(* IEC 61131-3 sources: LASAL/Class/ST151Base, 1 file *)

(* ---- ST151Base.st ---- *)
#define DEVICE_ID_ST151                                                    1086

#define ST151_ADDR_PDO_WRITE                                            16#0000
#define ST151_ADDR_PDO_READ                                             16#0038
#define ST151_ADDR_SDO_1                                                16#0008
#define ST151_ADDR_SDO_2           (ST151_ADDR_SDO_1+sizeof(t_s_ConfigModule1))
#define ST151_ADDR_SDO_3                                (ST151_ADDR_PDO_READ+6)  //only read sdo!!!
#define ST151_ADDR_SDO_4           (ST151_ADDR_SDO_3+sizeof(t_s_ConfigModule3))
#define ST151_ADDR_SDO_5           (ST151_ADDR_SDO_4+sizeof(t_s_ConfigModule4))
#define ST151_ADDR_SDO_6           (ST151_ADDR_SDO_5+sizeof(t_s_ConfigModule5))

#define ST151_OSZI_ADDR_WRITE                                           16#0800
#define ST151_OSZI_ADDR_READ                                            16#0808
#define ST151_OSZI_ADDR_DATA                                            16#0820
#define ST151_OSZI_READPOINTER_OFFSET                                   16#0020
#define ST151_OSZI_ONE_PDOSIZE                                              126
#define ST151_OSZI_VALUES_DATA             (ST151_OSZI_ONE_PDOSIZE/sizeof(UINT))
#define ST151_OSZI_BUFFER_SIZE                                             1024
#define ST151_OSZI_MAX_SAMPLES             (ST151_OSZI_BUFFER_SIZE/sizeof(UINT))
#define ST151_OSZI_MAX_PDOREAD   ((ST151_OSZI_BUFFER_SIZE/ST151_OSZI_ONE_PDOSIZE)+1)

// in MHz
#define ST151_FREQUENCY_MHZ                             125
// in Hz
#define ST151_FREQUENCY_HZ   (ST151_FREQUENCY_MHZ * 1000000)

#define ST151_SDO_RESPONSE_TIMEOUT   (SDIAS_SDO_TIMEOUT * 2)
#define ST151_SDO_MAX_RETRYS                              3

#define ST151_MAXFREQUENCY_OUT                   2_000_000 // 2Mhz/64 max frequency of module output
#define ST151_MAXSTEPPING_MODES                          6
#define ST151_FREQLIMITS_TABLESIZE      (ST151_MAXSTEPPING_MODES*sizeof(UDINT)*2)

#define ST151_MAX_ALLOWED_PERCENT                      100 // maximum value for percent value
#define ST151_BLANKING_TIME                             10 // minimum on time of pwm (*20ns)

#define ST151_CYCLICREFRESHDATA_TIME                   200 // time to refresh asynchrone values
#define ST151_INVALID_VALUE                   16#8000_0010 // invalid value for server
#define ST151_AUTOSET_FREQUENCYLIMIT          16#0000_0000 // value for autoset limit
#define ST151_DEACTIVATE_FREQUENCYLIMIT       16#FFFF_FFFF // value for deactivate limit

#define ST151_MAX_ALLOWED_CURRENT                     5000 // max allowed current (5A) in mA, from h-bridge according to hw-documentation
#define ST151_MAX_ALLOWED_CHOPPEROFFTIME              2500 // max allowed chopper off time in 20ns steps
#define ST151_MIN_ALLOWED_CHOPPEROFFTIME              1500 // min allowed chopper off time in 20ns steps
#define ST151_STALL_CURRENT_LIMIT                     1000 // calculation for stall current in permille
#define ST151_CURRENTOFFSETADJUST_MAX                  250 // maximum current offset adjust in mA
#define ST151_CURRENTOFFSETADJUST_MIN                 -250 // minimum current offset adjust in mA

//pll settings
#define ST151_SYNC_OUT_ID                             16#03
#define ST151_PLL_OFFSET                             16#140
#define ST151_PLL_CONTROL               (ST151_PLL_OFFSET+8)

#define ST151_ERROR_BITMASK_STATE_WORD               0x013E
#define ST151_ERROR_BITMASK_EXTENDED_STATE_WORD      0xFF3E

(*!
<Class
	Name               = "ST151Base"
	Revision           = "1.2"
	RealtimeTask       = "false"
	CyclicTask         = "false"
	BackgroundTask     = "false"
	Sigmatek           = "true"
	OSInterface        = "false"
	HighPriority       = "false"
	Automatic          = "false"
	UpdateMode         = "Prescan"
	IconPath           = ".\Class\s-dias.ico"
	SharedCommandTable = "true"
	Objectsize         = "(910,120)"
	Comment            = "SDIAS Stepper Module (1x Motor Out max. 5A, 2x Digital In 24V, 2x STO Enable 24V, 1x Incremental Encoder Input, 1x Regen Resistor)">
	<Channels>
		<Server Name="ActPosition" Visualized="true" Initialize="false" WriteProtected="true" Retentive="false" Comment="Actual internal Step-Position as 64 micro step."/>
		<Server Name="ActRegenResistorLoad" Visualized="true" Initialize="false" WriteProtected="true" Retentive="false" Comment="Actual load of regen resistor in xxx [%].&#13;&#10;If the value is never refreshed it shows -2 147 483 632.&#13;&#10;- Value is read asynchronous"/>
		<Server Name="AxError" Visualized="true" Initialize="false" WriteProtected="true" Retentive="false" Comment="Shows a fault of power-stage.&#13;&#10;(eg. over temperature, over current, power not connected)"/>
		<Server Name="ChopperOffTime" Visualized="true" Initialize="true" DefValue="1562" WriteProtected="false" Retentive="false" Comment="Set fixed off-time of the PWM  [20ns steps].&#13;&#10;If the value is changed, it is transferred asynchronously to the module.&#13;&#10;Valid range is from 1500 up to 2500."/>
		<Server Name="ChopperOnTimeMin" Visualized="true" Initialize="true" DefValue="180" WriteProtected="false" Retentive="false" Comment="Set minimum on-time of the PWM  [20ns steps].&#13;&#10;If the value is changed, it is transferred asynchronously to the module.&#13;&#10;Valid range is from 0 up to 2500."/>
		<Server Name="ControlWord" Visualized="true" Initialize="false" WriteProtected="false" Retentive="false" Comment="SwitchOn + Enable: Enable Motor&#13;&#10;ResetFault: Quit Error&#13;&#10;Bit12 ManufactureSpec1: current increase allowed"/>
		<Server Name="CurrentIncrease" Visualized="true" Initialize="true" DefValue="1" WriteProtected="false" Retentive="false" Comment="allow sqrt(2) current increase in halfstep mode&#13;&#10;&#13;&#10;in microstep mode the increase is always active"/>
		<Server Name="CurrentOffsetAdjBridge1" Visualized="true" Initialize="true" DefValue="100" WriteProtected="false" Retentive="false" Comment="!This setting has no effect if the version of the module is &gt;= HW2.0X1.4!&#13;&#10;&#13;&#10;Set current offset adjustment for bridge in [mA].&#13;&#10;Valid range is from -250 to 250 and default value is 100."/>
		<Server Name="CurrentOffsetAdjBridge2" Visualized="true" Initialize="true" DefValue="100" WriteProtected="false" Retentive="false" Comment="!This setting has no effect if the version of the module is &gt;= HW2.0X1.4!&#13;&#10;&#13;&#10;Set current offset adjustment for bridge in [mA].&#13;&#10;Valid range is from -250 to 250 and default value is 100."/>
		<Server Name="Enable" Visualized="true" Initialize="false" WriteProtected="false" Retentive="false" Comment="Enable stepper output.&#13;&#10;0 .. disabled&#13;&#10;1 .. enabled"/>
		<Server Name="EnableSteps" Visualized="true" Initialize="true" DefValue="2#1000111" WriteProtected="false" Retentive="false" Comment="Enable or disable microstepping modes. The full step mode cannot be deactivated.&#13;&#10;Bit1 .. Fullstep mode&#13;&#10;Bit2 .. Halfstep mode&#13;&#10;Bit3 .. Microstepping mode 4&#13;&#10;Bit4 .. Microstepping mode 8&#13;&#10;Bit5 .. Microstepping mode 16&#13;&#10;Bit6 .. Microstepping mode 32&#13;&#10;Bit7 .. Microstepping mode 64"/>
		<Server Name="EncoderPosition" Visualized="true" Initialize="false" WriteProtected="true" Retentive="false" Comment="Actual position of encoder."/>
		<Server Name="ErrorInfo" Visualized="true" Initialize="false" WriteProtected="true" Retentive="false" Comment="Shows errors from hardware. Errors above Bit 16 are refreshed at cyclic task over &quot;RefreshValues&quot; server.&#13;&#10;Bit 1: reserved&#13;&#10;Bit 2: Fault (Bridge not ok)&#13;&#10;Bit 3: Temperature  not ok&#13;&#10;Bit 4: Over current&#13;&#10;Bit 5: STO switch off (en1/en2)&#13;&#10;Bit 6: STO test switch off (negative test during operation)&#13;&#10;Bit 7: reserved&#13;&#10;Bit 8: reserved&#13;&#10;Bit 9: Brake chopper over current (disable brake chopper) &#13;&#10;Bit 10: reserved&#13;&#10;Bit 11: reserved&#13;&#10;Bit 12: reserved&#13;&#10;Bit 13: reserved&#13;&#10;Bit 14: reserved&#13;&#10;Bit 15: reserved&#13;&#10;Bit 16: reserved&#13;&#10;&#13;&#10;refreshed asynchrone:&#13;&#10;Bit 17: Regen resistor load warning&#13;&#10;Bit 18: Over temperature warning&#13;&#10;Bit 19: Over temperature failure (disable drive)&#13;&#10;Bit 20: Over current failure GND (disable drive)&#13;&#10;Bit 21: Over current failure Bridge 1 (disable drive)&#13;&#10;Bit 22: Over current failure Bridge 2 (disable drive)&#13;&#10;Bit 23: Regen resistor load threshold bridge (disable bridge)&#13;&#10;Bit 24: Regen resistor load error threshold resistor (disable resistor)&#13;&#10;Bit 25: Bridge voltage too low&#13;&#10;Bit 26: Bridge voltage too high&#13;&#10;Bit 27: External Enable 1 (STO) not ok&#13;&#10;Bit 28: External Enable 2 (STO) not ok&#13;&#10;Bit 29: Safety start up status test not ok&#13;&#10;Bit 30: Motor enable error&#13;&#10;Bit 31: Three time sync in lost&#13;&#10;Bit 32: Safe Ramp down pending"/>
		<Server Name="ErrorQuit" Visualized="true" Initialize="false" WriteProtected="false" Retentive="false" Comment="quits error if server &quot;Error&quot; is set"/>
		<Server Name="ExtendedStateWord" Visualized="true" Initialize="false" WriteProtected="true" Retentive="false" Comment="Shows the extended motor state word.&#13;&#10;- Value is read asynchronous&#13;&#10;Bit 1 : Zero Position (Input)&#13;&#10;Bit 2 : Over temperature warning&#13;&#10;Bit 3 : Over temperature failure (disable drive)&#13;&#10;Bit 4 : Over current failure GND (disable drive)&#13;&#10;Bit 5 : Over current failure Bridge 1 (disable drive)&#13;&#10;Bit 6 : Over current failure Bridge 2 (disable drive)&#13;&#10;Bit 7 : 5V Incremental encoder ok&#13;&#10;Bit 8 : reserved&#13;&#10;Bit 9 : Bridge voltage too low&#13;&#10;Bit 10: Bridge voltage too high&#13;&#10;Bit 11: External Enable 1 (STO)&#13;&#10;Bit 12: External Enable 2 (STO)&#13;&#10;Bit 13: Safety start up status test ok&#13;&#10;Bit 14: Motor enable error&#13;&#10;Bit 15: Three time sync in lost&#13;&#10;Bit 16: Safe Ramp down pending"/>
		<Server Name="ExternalEnable1" Visualized="true" Initialize="false" WriteProtected="true" Retentive="false" Comment="State of External Enable  (STO).&#13;&#10;If the value is never refreshed it shows -2 147 483 632.&#13;&#10;- Value is read asynchronous&#13;&#10;0 .. off&#13;&#10;1 .. on&#13;&#10;"/>
		<Server Name="ExternalEnable2" Visualized="true" Initialize="false" WriteProtected="true" Retentive="false" Comment="State of External Enable  (STO).&#13;&#10;If the value is never refreshed it shows -2 147 483 632.&#13;&#10;- Value is read asynchronous&#13;&#10;0 .. off&#13;&#10;1 .. on&#13;&#10;"/>
		<Server Name="FastDecayTime" Visualized="true" Initialize="true" DefValue="200" WriteProtected="false" Retentive="false" Comment="Set Fast Decay time [20ns steps].&#13;&#10;If the value is changed, it is transferred asynchronously to the module.&#13;&#10;Must be smaller than chopper off time!"/>
		<Server Name="FastDecayTimeFallingStep" Visualized="true" Initialize="true" DefValue="600" WriteProtected="false" Retentive="false" Comment="Set Fast Decay time for falling step [20ns steps].&#13;&#10;If the value is changed, it is transferred asynchronously to the module.&#13;&#10;Must be smaller than chopper off time!"/>
		<Server Name="FrequLimitDecrease16to32" Visualized="true" Initialize="true" DefValue="0" WriteProtected="false" Retentive="false" Comment="Set Frequency stepping mode limit if frequence is decreased.&#13;&#10;If the value is changed, it is transferred asynchronously to the module.&#13;&#10;If value is set to 0 the limit is automatically set."/>
		<Server Name="FrequLimitDecrease1to2" Visualized="true" Initialize="true" DefValue="0" WriteProtected="false" Retentive="false" Comment="Set Frequency stepping mode limit if frequence is decreased.&#13;&#10;If the value is changed, it is transferred asynchronously to the module.&#13;&#10;If value is set to 0 the limit is automatically set."/>
		<Server Name="FrequLimitDecrease2to4" Visualized="true" Initialize="true" DefValue="0" WriteProtected="false" Retentive="false" Comment="Set Frequency stepping mode limit if frequence is decreased.&#13;&#10;If the value is changed, it is transferred asynchronously to the module.&#13;&#10;If value is set to 0 the limit is automatically set."/>
		<Server Name="FrequLimitDecrease32to64" Visualized="true" Initialize="true" DefValue="0" WriteProtected="false" Retentive="false" Comment="Set Frequency stepping mode limit if frequence is decreased.&#13;&#10;If the value is changed, it is transferred asynchronously to the module.&#13;&#10;If value is set to 0 the limit is automatically set."/>
		<Server Name="FrequLimitDecrease4to8" Visualized="true" Initialize="true" DefValue="0" WriteProtected="false" Retentive="false" Comment="Set Frequency stepping mode limit if frequence is decreased.&#13;&#10;If the value is changed, it is transferred asynchronously to the module.&#13;&#10;If value is set to 0 the limit is automatically set."/>
		<Server Name="FrequLimitDecrease8to16" Visualized="true" Initialize="true" DefValue="0" WriteProtected="false" Retentive="false" Comment="Set Frequency stepping mode limit if frequence is decreased.&#13;&#10;If the value is changed, it is transferred asynchronously to the module.&#13;&#10;If value is set to 0 the limit is automatically set."/>
		<Server Name="FrequLimitIncrease16to8" Visualized="true" Initialize="true" DefValue="20000" WriteProtected="false" Retentive="false" Comment="Set Frequency stepping mode limit if frequence is increased.&#13;&#10;If the value is changed, it is transferred asynchronously to the module.&#13;&#10;"/>
		<Server Name="FrequLimitIncrease2to1" Visualized="true" Initialize="true" DefValue="50000" WriteProtected="false" Retentive="false" Comment="Set Frequency stepping mode limit if frequence is increased.&#13;&#10;If the value is changed, it is transferred asynchronously to the module.&#13;&#10;"/>
		<Server Name="FrequLimitIncrease32to16" Visualized="true" Initialize="true" DefValue="10000" WriteProtected="false" Retentive="false" Comment="Set Frequency stepping mode limit if frequence is increased.&#13;&#10;If the value is changed, it is transferred asynchronously to the module.&#13;&#10;"/>
		<Server Name="FrequLimitIncrease4to2" Visualized="true" Initialize="true" DefValue="40000" WriteProtected="false" Retentive="false" Comment="Set Frequency stepping mode limit if frequence is increased.&#13;&#10;If the value is changed, it is transferred asynchronously to the module.&#13;&#10;"/>
		<Server Name="FrequLimitIncrease64to32" Visualized="true" Initialize="true" DefValue="5000" WriteProtected="false" Retentive="false" Comment="Set Frequency stepping mode limit if frequence is increased.&#13;&#10;If the value is changed, it is transferred asynchronously to the module.&#13;&#10;"/>
		<Server Name="FrequLimitIncrease8to4" Visualized="true" Initialize="true" DefValue="30000" WriteProtected="false" Retentive="false" Comment="Set Frequency stepping mode limit if frequence is increased.&#13;&#10;If the value is changed, it is transferred asynchronously to the module.&#13;&#10;"/>
		<Server Name="HBridgeTemperature" Visualized="true" Initialize="false" WriteProtected="true" Retentive="false" Comment="actual Temperature in xx.x [°C]&#13;&#10;If the value is never refreshed it shows -2 147 483 632.&#13;&#10;- Value is read asynchronous."/>
		<Server Name="HBridgeVoltage" Visualized="true" Initialize="false" WriteProtected="true" Retentive="false" Comment="Actual Voltage in xx.xx [V].&#13;&#10;If the value is never refreshed it shows -2 147 483 632.&#13;&#10;- Value is read asynchronous"/>
		<Server Name="HWEnableSoftwareRampdown" Visualized="true" Initialize="true" WriteProtected="false" Retentive="false" Comment=" 0 ... HardwareRampdown&#13;&#10; 1 ... SoftwareRampdown"/>
		<Server Name="HWRampdownDeltaFrequency" Visualized="true" Initialize="true" DefValue="40" WriteProtected="false" Retentive="false" Comment="If the enable-signal is lost the output frequency is decreased by HWRampdownDeltaFrequency every HWRampdownDeltaTime"/>
		<Server Name="HWRampdownDeltaTime" Visualized="true" Initialize="true" DefValue="1" WriteProtected="false" Retentive="false" Comment="[20ns steps]&#13;&#10;If the enable-signal is lost the output frequency is decreased by HWRampdownDeltaFrequency every HWRampdownDeltaTime"/>
		<Server Name="Input1" Visualized="true" Initialize="false" WriteProtected="true" Retentive="false" Comment="first digital input"/>
		<Server Name="Input1LatchedFalling" Visualized="true" Initialize="false" WriteProtected="true" Retentive="false" Comment="latched falling edge of first digital input&#13;&#10;signal will stay until read-method is called"/>
		<Server Name="Input1LatchedRising" Visualized="true" Initialize="false" WriteProtected="true" Retentive="false" Comment="latched rising edge of first digital input&#13;&#10;signal will stay until read-method is called"/>
		<Server Name="Input2" Visualized="true" Initialize="false" WriteProtected="true" Retentive="false" Comment="second digital input"/>
		<Server Name="Input2LatchedFalling" Visualized="true" Initialize="false" WriteProtected="true" Retentive="false" Comment="latched falling edge of second digital input&#13;&#10;signal will stay until read-method is called"/>
		<Server Name="Input2LatchedRising" Visualized="true" Initialize="false" WriteProtected="true" Retentive="false" Comment="latched rising edge of second digital input&#13;&#10;signal will stay until read-method is called"/>
		<Server Name="LatchPositionEncoderZeroPulse" Visualized="true" Initialize="false" WriteProtected="true" Retentive="false" Comment="Latched position of encoder zero pulse."/>
		<Server Name="LatchPositionInput1Falling" Visualized="true" Initialize="false" WriteProtected="true" Retentive="false" Comment="Latched position of falling edge of input 1."/>
		<Server Name="LatchPositionInput1Rising" Visualized="true" Initialize="false" WriteProtected="true" Retentive="false" Comment="Latched position of rising edge of input 1."/>
		<Server Name="LatchPositionInput2Falling" Visualized="true" Initialize="false" WriteProtected="true" Retentive="false" Comment="Latched position of falling edge of input 2."/>
		<Server Name="LatchPositionInput2Rising" Visualized="true" Initialize="false" WriteProtected="true" Retentive="false" Comment="Latched position of rising edge of input 2."/>
		<Server Name="MaxCurrent" Visualized="true" Initialize="true" WriteProtected="false" Retentive="false" Comment="Set maximum output current [mA] (effectiv value) as init value.&#13;&#10;If value is changed it is written asynchronosly.&#13;&#10;If the value is changed, it is transferred asynchronously to the module.&#13;&#10;Valid range is from 0 up to 5000."/>
		<Server Name="Online" Visualized="true" Initialize="false" WriteProtected="true" Retentive="false" Comment="Shows if hardware is ready.&#13;&#10;0 .. not ready&#13;&#10;1 .. ready"/>
		<Server Name="RefreshValues" Visualized="true" Initialize="true" WriteProtected="false" Retentive="false" Comment="Set refresh of asynchrone values&#13;&#10; 0 .. do not refresh values&#13;&#10; 1 .. do cyclic refresh of values (every 200ms)&#13;&#10; 2 .. refresh values once"/>
		<Server Name="SetFreqOut" Visualized="true" Initialize="false" WriteProtected="false" Retentive="false" Comment="Frequency in Hz of one Microstep [1/64 Hz]&#13;&#10;64 Microsteps = 1 Fullstep"/>
		<Server Name="StateWord" Visualized="true" Initialize="false" WriteProtected="true" Retentive="false" Comment="Statusword with DS402 Standard :&#13;&#10;Bit1  .. ReadyToSwitchOn&#13;&#10;Bit2  .. SwitchedOn&#13;&#10;Bit3  .. OperationEnabled&#13;&#10;Bit4  .. Fault&#13;&#10;Bit5  .. VoltageDisabled&#13;&#10;Bit6  .. QuickStop&#13;&#10;Bit7  .. SwitchOnDisabled&#13;&#10;Bit8  .. Warning&#13;&#10;Bit9  .. ManufactureSpecific1&#13;&#10;Bit10 .. Remote&#13;&#10;Bit11 .. TargetReached&#13;&#10;Bit12 .. InternalLimitActive&#13;&#10;Bit13 .. OperationModeSpecific1&#13;&#10;Bit14 .. OperationModeSpecific2&#13;&#10;Bit15 .. Manufacture Specific2&#13;&#10;Bit16 .. Manufacture Specific3"/>
		<Server Name="TargetFreqOut" Visualized="true" Initialize="false" WriteProtected="false" Retentive="false" Comment="Set desired motor frequency in [1/64 Hz].&#13;&#10;This value is needed for adaptive Microstepping calculation.&#13;&#10;64 Microsteps = 1 Fullstep&#13;&#10;-1 .. feature is deactivated."/>
		<Server Name="VoltageOKEncoder" Visualized="true" Initialize="false" WriteProtected="true" Retentive="false" Comment="Shows state of voltage supply of encoder.&#13;&#10;If the value is never refreshed it shows -2 147 483 632.&#13;&#10;- Value is read asynchronous&#13;&#10;0 .. Error at power supply.&#13;&#10;1 .. OK"/>
		<Server Name="ZPuls" Visualized="true" Initialize="false" WriteProtected="true" Retentive="false" Comment="It is 1 if incremental encoder zero position is passed."/>
		<Server Name="ZPulsLatched" Visualized="true" Initialize="false" WriteProtected="true" Retentive="false" Comment="It is 1 if incremental encoder zero position is passed, a read resets the server"/>
		<Client Name="ABCountMode" Required="true" Internal="false" DefValue="1" Comment="Set A/B count mode if &quot;1 edge&quot; sampling is activated, as init value.&#13;&#10;0 .. A pulses, B direction&#13;&#10;1 .. true A/B (default)"/>
		<Client Name="CompModeVST" Required="true" Internal="false" DefValue="0" Comment="Set Compatibility mode to VST01x as init value.&#13;&#10;0 .. Frequency as 64 microsteps - default&#13;&#10;1 .. Frequency as 32 microsteps&#13;&#10;This setting affects all &quot;FrequencyLimitsIncrease&quot;, &quot;FrequencyLimitsDecrease&quot;, &quot;SetFreqOut&quot;, &quot;ActPosition&quot;, &#13;&#10;&quot;TargetFreqOut&quot; server and the &quot;Latched Position&quot; server if LatchType is latch virtual counter."/>
		<Client Name="EnableRegenResistor" Required="true" Internal="false" DefValue="0" Comment="Enable external regen resistor.&#13;&#10;0 .. disabled&#13;&#10;1 .. enabled"/>
		<Client Name="EncMode" Required="true" Internal="false" DefValue="0" Comment="Mode of the Incremental Encoder as init value.&#13;&#10;0 .. TTL&#13;&#10;1 .. RS422&#13;&#10;"/>
		<Client Name="EncoderSampling" Required="true" Internal="false" DefValue="3" Comment="Sampling of the Incremental Encoder.&#13;&#10;0 .. Encoder off&#13;&#10;1 .. 1-edge&#13;&#10;2 .. 2-edge&#13;&#10;3 .. 4-edge&#13;&#10;"/>
		<Client Name="InvertEncoder" Required="true" Internal="false" DefValue="0" Comment="Counting direction of the encoder as initvalue.&#13;&#10;0 .. Phase B non-inverted&#13;&#10;1 .. Phase B inverted&#13;&#10;&#13;&#10;"/>
		<Client Name="InvertZeroPosition" Required="true" Internal="false" DefValue="0" Comment="Inverts server ZPulse as initvalue.&#13;&#10;0..normal &#13;&#10;1..inverted&#13;&#10;"/>
		<Client Name="LatchType" Required="true" Internal="false" DefValue="0" Comment="0 .. latch virtual counter&#13;&#10;1 .. latch incremental encoder&#13;&#10;as initvalue"/>
		<Client Name="LoadThresholdBridge" Required="true" Internal="false" DefValue="90" Comment="Set threshold value for regen resistor load [%] to switch off bridge, as init value.&#13;&#10;If this limit is reached, the bridge is switched off.&#13;&#10;Valid Range is 0 up to 100% and default value is 90%."/>
		<Client Name="LoadThresholdResistor" Required="true" Internal="false" DefValue="100" Comment="Set threshold value for regen resistor load [%] to switch external resistor off, as init value. &#13;&#10;If this limit is reached, the bridge and the regen resistor is switched off.&#13;&#10;Valid Range is 0 up to 100% and default value is 100%."/>
		<Client Name="LoadThresholdWarning" Required="true" Internal="false" DefValue="80" Comment="Set threshold value for regen resistor load [%] to set the warning bit, as init value.&#13;&#10;Valid Range is 0 up to 100% and default value is 80%."/>
		<Client Name="RatedMaxPower" Required="true" Internal="false" DefValue="1000" Comment="Set value for rated maximum Power of regen resistor in [1/10 W] as init value.&#13;&#10;Value is needed for capacity calculation of resistor.&#13;&#10;Valid range is from 1 up to 65535."/>
		<Client Name="RegenResistance" Required="true" Internal="false" DefValue="150" Comment="Set resistance of regen resistor in [1/10 Ohm] as init value.&#13;&#10;Value is needed for capacity calculation of resistor.&#13;&#10;Valid range is from 1 up to 65535."/>
		<Client Name="StallCurrentReduction" Required="true" Internal="false" DefValue="0" Comment="Value to reduce MaxCurrent for the Stop Position [0,1%] as init value. &#13;&#10;Defaultvalue: 0 (no reduction in the stop position)&#13;&#10;Range: 0 - 1000 (0-100%)&#13;&#10;Stop Position means, the value of the server SetFreqOut is lower than the StallCurrentWindow, &#13;&#10;which can be set with StallCurrentWindow and is 0 by default."/>
		<Client Name="StallCurrentWindow" Required="true" Internal="false" DefValue="0" Comment="Set a window in which the StallCurrentReduction setting is active as init value.&#13;&#10;Valid range is from 0 up to 65535."/>
		<Client Name="SteppingHysteresis" Required="true" Internal="false" DefValue="64" Comment="Set automatically stepping hysterese in [1/64 Hz] if the value for decrease limit is zero as init value.&#13;&#10;This value is substracted from the corresponding increase limit value and set for the decrease limit."/>
		<Client Name="toFreqLimitTable" Required="false" Internal="false"/>
		<Client Name="UseOszi" Required="true" Internal="false" DefValue="0" Comment="Activate oszi function of modul as init value.&#13;&#10;To use the Oszi function, the methods &quot;StartMeasure ()&quot; and &quot;GetMeasureState ()&quot; must be used.&#13;&#10;&#13;&#10;0 .. deactivated&#13;&#10;1 .. activated"/>
	</Channels>
	<Separators>
		<Servers>
			<SepChn Position="1"/>
			<SepChn Position="16"/>
			<SepChn Position="50"/>
		</Servers>
		<Clients>
			<SepChn Position="6"/>
		</Clients>
	</Separators>
	<RevDoku>
		<Owner Company="Sigmatek" Author="PieSte"/>
		<Dokumentation Revision="1.2" Date="31.07.2018" Author="RamAnd" Company="Sigmatek" Description="LASAL Hardware Description (.lhd) file has been updated.&#13;&#10;Removed initialize flag from server TargetFreqOut."/>
		<Dokumentation Revision="1.1" Date="01.02.2018" Author="ZoePat" Company="Sigmatek" Description="An error has been fixed if server settings were written in the init()."/>
		<Dokumentation Revision="1.0" Date="22.11.2017" Author="ZoePat" Company="Sigmatek" Description="first release version."/>
	</RevDoku>
	<Network Name="ST151Base">
		<!-- List of Components in this network -->
		<Components>
			<Object
				Name       = "_base"
				Class      = "SdiasBase"
				Position   = "(218,120)"
				Visualized = "true">
				<Channels>
					<Server Name="ClassState"/>
					<Server Name="DeviceID"/>
					<Server Name="FPGAVersion"/>
					<Server Name="HwVersion"/>
					<Server Name="LEDControl" Value="0"/>
					<Server Name="RetryCounter"/>
					<Server Name="SDOState"/>
					<Server Name="SerialNo"/>
					<Client Name="Place" Value="0"/>
					<Client Name="Required" Value="1"/>
					<Client Name="SdiasIn"/>
					<Client Name="ToStdLib"/>
				</Channels>
			</Object>
		</Components>
		<Comments>
		</Comments>
		<!-- List of Connections in this network -->
		<Connections>
			<Connection Source="this.ClassState" Destination="_base.ClassState" Vertices="(804,210),(632,210),"/>
			<Connection Source="this.DeviceID" Destination="_base.DeviceID" Vertices="(804,270),(632,270),"/>
			<Connection Source="this.FPGAVersion" Destination="_base.FPGAVersion" Vertices="(804,330),(632,330),"/>
			<Connection Source="this.SerialNo" Destination="_base.SerialNo" Vertices="(804,450),(632,450),"/>
			<Connection Source="this.RetryCounter" Destination="_base.RetryCounter" Vertices="(804,510),(632,510),"/>
			<Connection Source="this.LEDControl" Destination="_base.LEDControl" Vertices="(804,570),(632,570),"/>
			<Connection Source="_base.SdiasIn" Destination="this.SdiasIn" Vertices="(218,210),(38,210),"/>
			<Connection Source="_base.Place" Destination="this.Place" Vertices="(218,270),(38,270),"/>
			<Connection Source="_base.Required" Destination="this.Required" Vertices="(218,330),(38,330),"/>
			<Connection Source="this.HwVersion" Destination="_base.HwVersion" Vertices="(804,390),(632,390),"/>
			<Connection Source="this.SDOState" Destination="_base.SDOState" Vertices="(804,630),(632,630),"/>
		</Connections>
		<!-- Headerfiles -->
		<Options>
		</Options>
	</Network>
</Class>
*)
#pragma using SdiasBase

ST151Base : CLASS
: SdiasBase
	TYPE
	  a_uiOsziValues : ARRAY [0..ST151_OSZI_VALUES_DATA-1] OF UINT;
	  bd_EnabledFreqLimit : BDINT  //! <Type Public="true" Name="bd_EnabledFreqLimit"/>
	  [
	    1 FullStep,
	    2 HalfStep,
	    3 MicroStepping4,
	    4 MicroStepping8,
	    5 MicroStepping16,
	    6 MicroStepping32,
	    7 MicroStepping64,
	    8 Bit8,
	    9 Bit9,
	    10 Bit10,
	    11 Bit11,
	    12 Bit12,
	    13 Bit13,
	    14 Bit14,
	    15 Bit15,
	    16 Bit16,
	    17 Bit17,
	    18 Bit18,
	    19 Bit19,
	    20 Bit20,
	    21 Bit21,
	    22 Bit22,
	    23 Bit23,
	    24 Bit24,
	    25 Bit25,
	    26 Bit26,
	    27 Bit27,
	    28 Bit28,
	    29 Bit29,
	    30 Bit30,
	    31 Bit31,
	    32 Bit32,
	  ];
	  bd_ExtendedStateWord : BDINT  //! <Type Public="true" Name="bd_ExtendedStateWord"/>
	  [
	    1 ZeroPosition,
	    2 OverTempWarning,
	    3 OverTempFailure,
	    4 OverCurrentFailureGND,
	    5 OverCurrentFailureBridge1,
	    6 OverCurrentFailureBridge2,
	    7 Encoder5VOk,
	    8 Bit8,
	    9 BridgeVoltageTooLow,
	    10 BridgeVoltageTooHigh,
	    11 ExternEnableSTO1,
	    12 ExternEnableSTO2,
	    13 SafetyStartUpOK,
	    14 MotorEnableError,
	    15 ThreeTimeSyncInLost,
	    16 SafeRampDownPending,
	    17 LoadWarning,
	    18 LoadDisableBridge,
	    19 LoadDisableResistor,
	    20 Bit20,
	    21 Bit21,
	    22 Bit22,
	    23 Bit23,
	    24 Bit24,
	    25 Bit25,
	    26 Bit26,
	    27 Bit27,
	    28 Bit28,
	    29 Bit29,
	    30 Bit30,
	    31 Bit31,
	    32 Bit32,
	  ];
	  e_ActStepMode :
	  (
	    Microstepping_1,
	    Microstepping_2,
	    Microstepping_4,
	    Microstepping_8,
	    Microstepping_16,
	    Microstepping_32,
	    Microstepping_64
	  )$UDINT;
	  t_StatusWord : BINT
	  [
	    1 MotorEnabled,
	    2 Fault,
	    3 TemperatureOk,
	    4 OverCurrent,
	    5 STOSwitchOff,
	    6 STOTestSwitchOff,
	    7 STOReadyRestart,
	    8 ReadyToSwitchOn,
	    9 BrakeChopperOverCurrentLatch,
	    10 LatchIncZero,
	    11 LatchDigIn1Rise,
	    12 LatchDigIn1Fall,
	    13 LatchDigIn2Rise,  //! <Type Comment="Low bit of failure state depending on InternalLimitActive bit&#13;&#10;&#13;&#10;Meaning:&#13;&#10;2#00...No failure&#13;&#10;2#01...Overtemperature failure&#13;&#10;2#10...Overcurrent failure" Name="t_StatusWord.LatchDigIn2Rise"/>
	    14 LatchDigIn2Fall,  //! <Type Comment="High bit of failure state depending on InternalLimitActive bit&#13;&#10;&#13;&#10;Meaning:&#13;&#10;2#00...No failure&#13;&#10;2#01...Overtemperature failure&#13;&#10;2#10...Overcurrent failure" Name="t_StatusWord.LatchDigIn2Fall"/>
	    15 DigIn1,  //! <Type Comment="Low bit of failure state depending on InternalLimitActive bit&#13;&#10;&#13;&#10;Meaning:&#13;&#10;2#00...No failure&#13;&#10;2#01...Overtemperature failure&#13;&#10;2#10...Overcurrent failure" Name="t_StatusWord.DigIn1"/>
	    16 DigIn2,  //! <Type Comment="High bit of failure state depending on InternalLimitActive bit&#13;&#10;&#13;&#10;Meaning:&#13;&#10;2#00...No failure&#13;&#10;2#01...Overtemperature failure&#13;&#10;2#10...Overcurrent failure" Name="t_StatusWord.DigIn2"/>
	  ];
#pragma pack(push, 1)
	  t_s_ReadData : STRUCT
	    StateWord : t_StatusWord;
	    ActPos : UINT;
	    IncrementalEncoderValue : UINT;
	  END_STRUCT;
#pragma pack(pop)
	  t_ControlWord : BINT
	  [
	    1 SwitchOn,
	    2 FaultReset,
	    3 CurrentDropEnable,
	    4 CurrentIncrease,
	    5 HWEnableSofwareRampdownToggleBit,
	    6 QuitSTOOff,
	    7 RegenResistorEnable,
	    8 RegenResistorFaultReset,
	    9 SwitchMaxCurrent,  //! <Type Comment="0 .. internal counter&#13;&#10;1 .. incremental encoder" Name="t_ControlWord.SwitchMaxCurrent"/>
	    10 EnableStep64,
	    11 EnableStep32,
	    12 EnableStep16,
	    13 EnableStep8,
	    14 EnableStep4,
	    15 EnableHalfStep,
	    16 EnableFullStep,
	  ];
#pragma pack(push, 1)
	  t_s_WriteData : STRUCT
	    StepFrequencyReg : DINT;
	    ControlWord : t_ControlWord;
	  END_STRUCT;
#pragma pack(pop)
#pragma pack(push, 1)
	  t_Accesses : STRUCT
	    pReadData : ^t_s_ReadData;
	    pWriteData : ^t_s_WriteData;
	    sWriteData : t_s_WriteData;
	  END_STRUCT;
#pragma pack(pop)
#pragma pack(push, 1)
	  t_s_ControlAccess : STRUCT
	    AccessHandle : UDINT;
	    pControlByte : t_SDIAS_pControlByte;
	    pStateByte : t_SDIAS_pStateByte;
	  END_STRUCT;
#pragma pack(pop)
#pragma pack(push, 1)
	  t_s_OsziWrite : STRUCT
	    SamplesAfterTrigger : UINT;
	    TriggerLevel : UINT;
	    SampleTimePrescaler : UINT;
	    TriggerChannelSelect : USINT;
	    ControlOszi : BSINT
	    [
	      1 StartTriggering,
	      2 CancelTrigger,
	      3 RisingEdge,
	      4 FallingEdge,
	      5 Force,
	      6 Bit6,
	      7 Bit7,
	      8 Bit8,
	    ];
	  END_STRUCT;
#pragma pack(pop)
#pragma pack(push, 1)
	  t_s_OsziRead : STRUCT
	    SizeOfRam : UDINT;
	    PointerOnLastSampleData : HDINT;
	    StateOszi : BSINT
	    [
	      1 Ready,
	      2 Triggered,
	      3 BufferOverflow,
	      4 Bit4,
	      5 Bit5,
	      6 Bit6,
	      7 Bit7,
	      8 Bit8,
	    ];
	    NbrOfChAvailable : USINT;
	  END_STRUCT;
#pragma pack(pop)
#pragma pack(push, 1)
	  t_AccessesOszi : STRUCT
	    WriteHeaderControl : t_s_ControlAccess;
	    pWriteHeader : ^t_s_OsziWrite;
	    sWriteOszi : t_s_OsziWrite;
	    ReadHeaderControl : t_s_ControlAccess;
	    pReadHeader : ^t_s_OsziRead;
	    aReadDataControl : ARRAY [0..ST151_OSZI_MAX_PDOREAD-1] OF t_s_ControlAccess;
	    apOsziData : ARRAY [0..ST151_OSZI_MAX_PDOREAD-1] OF ^a_uiOsziValues;
	    uiSamplesAfterTrigger : UINT;
	    uiSamplesBeforeTrigger : UINT;
	    bDataReady : DINT;
	    bSplitBuffer : BOOL;
	    uiDatalength1 : UINT;
	    uiDatalength2 : UINT;
	    eOsziData :
	    (
	      _OsziDataIdle,
	      _OsziTriggerStart,
	      _OsziResetTrigger,
	      _OsziWait4Reset,
	      _OsziWait4Trigger,
	      _OsziDisableRead,
	      _OsziGetData,
	      _OsziWait4Data,
	      _OsziFinished
	    )$UDINT;
	    sLastOsziState : t_s_OsziRead;
	    aLastOsziData : ARRAY [0..ST151_OSZI_MAX_SAMPLES-1] OF UINT;
	    pLastEntryOsziData : ^UINT;
	    pFirstEntryOsziData : ^UINT;
	    pToExternData : ^void;
	    usOsziTriggerOffset : USINT;
	    bMeasureStarted : BOOL;
	  END_STRUCT;
#pragma pack(pop)
	  t_bi_ReqSDOConfig : BINT
	  [
	    1 WriteConfigSDO1,
	    2 WriteConfigSDO2,
	    3 WriteConfigSDO3,
	    4 WriteConfigSDO4,
	    5 WriteConfigSDO5,
	    6 WriteConfigSDO6,
	    7 Bit7,
	    8 ReadConfigSDO1,
	    9 ReadConfigSDO2,
	    10 ReadConfigSDO3,
	    11 ReadConfigSDO4,
	    12 ReadConfigSDO5,
	    13 ReadConfigSDO6,
	    14 Bit14,
	    15 Bit15,
	    16 Bit16,
	  ];
	  t_bs_IsyncValue : BSINT
	  [
	    1 IncZero,
	    2 DigIn1Rise,
	    3 DigIn1Fall,
	    4 DigIn2Rise,
	    5 DigIn2Fall,
	  ];
	  t_e_InitSSW :
	  (
	    _ReadInitValuesFromModule,
	    _InitVariables,
	    _WriteConfigSDO,
	    _ReadConfigSDO,
	    _DisablePll,
	    _ReadPll,
	    _SetPll,
	    _Wait4FPGAReset,
	    _ActivateFPGA,
	    _Finish,
	    _InitError
	  )$UDINT;
	  t_e_SDOConfig :
	  (
	    _SDOConfig_Idle,
	    _SDOConfig_Write1,
	    _SDOConfig_Write2,
	    _SDOConfig_Write3,
	    _SDOConfig_Write4,
	    _SDOConfig_Write5,
	    _SDOConfig_Write6,
	    _SDOConfig_Read1,
	    _SDOConfig_Read2,
	    _SDOConfig_Read3,
	    _SDOConfig_Read4,
	    _SDOConfig_Read5,
	    _SDOConfig_Read6,
	    _SDOConfig_Finished,
	    _SDOConfig_Error
	  )$UDINT;
#pragma pack(push, 1)
	  t_EnabledFreqLimit : STRUCT
	    DecreaseFreq : bd_EnabledFreqLimit;
	    IncreaseFreq : bd_EnabledFreqLimit;
	  END_STRUCT;
#pragma pack(pop)
#pragma pack(push, 1)
	  t_FrequencyLimits : STRUCT
	    LimitDecrease : UDINT;  //! <Type Comment="save the higher limit" Name="t_FrequencyLimits.LimitDecrease"/>
	    LimitIncrease : UDINT;  //! <Type Comment="save the lower limit" Name="t_FrequencyLimits.LimitIncrease"/>
	  END_STRUCT;
#pragma pack(pop)
#pragma pack(push, 1)
	  t_LatchValues : STRUCT
	    uiISyncIncZeroOldCounter : UINT;
	    uiISyncDigIn1RiseOldCounter : UINT;
	    uiISyncDigIn1FallOldCounter : UINT;
	    uiISyncDigIn2RiseOldCounter : UINT;
	    uiISyncDigIn2FallOldCounter : UINT;
	    sdISyncIncZeroOldPosition : DINT;
	    sdISyncDigIn1RiseOldPosition : DINT;
	    sdISyncDigIn1FallOldPosition : DINT;
	    sdISyncDigIn2RiseOldPosition : DINT;
	    sdISyncDigIn2FallOldPosition : DINT;
	    uiLatchInputZero : DINT;
	    uiLatchInputDigIn1Rising : UINT;
	    uiLatchInputDigIn1Falling : UINT;
	    uiLatchInputDigIn2Rising : UINT;
	    uiLatchInputDigIn2Falling : UINT;
	    bsValidISyncValue : t_bs_IsyncValue;
	    bsActiveISyncValue : t_bs_IsyncValue;
	    bsLatchReaded : t_bs_IsyncValue;
	    bResetActiveSyncValue : BOOL;
	  END_STRUCT;
#pragma pack(pop)
#pragma pack(push, 1)
	  t_SyncOut : STRUCT
	    uiOffset : UINT;
	    usPeriodMulti : USINT;
	    bsSyncStartDelay : BSINT
	    [
	      1 SyncStartDelay1,
	      2 SyncStartDelay2,
	      3 SyncStartDelay3,
	      4 SyncStartDelay4,
	    ];
	    hsSyncOutID : HSINT;
	    bsControlState : BSINT
	    [
	      1 SyncEnable,
	      2 StartDelayEnable,
	      3 SyncSelector,
	    ];
	    uiReserved : UINT;
	  END_STRUCT;
#pragma pack(pop)
#pragma pack(push, 1)
	  t_PllRegister : STRUCT
	    udSystemPerTime : UDINT;
	    udSystemPerTimeMeasure : UDINT;
	    bsStateControlReg : BSINT
	    [
	      1 locked_res1,
	      2 unlocked_res2,
	      3 Soft_enable,
	      4 res3,
	      5 res4,
	      6 res5,
	      7 res6,
	      8 res7,
	    ];
	    usSystemPeriodeDividier : USINT;
	    bsCompDelay : BSINT
	    [
	    ];
	    usReserved : USINT;
	    SyncOut0 : t_SyncOut;
	  END_STRUCT;
#pragma pack(pop)
	  t_ResponseState :
	  (
	    _idle,
	    _wait,
	    _valid
	  )$UDINT;
#pragma pack(push, 1)
	  t_s_AdaptiveSteppingCalc : STRUCT
	    usIncreaseActStepsActivated : USINT;
	    aIncreaseLimitsArrayEntry : ARRAY [0..ST151_MAXSTEPPING_MODES] OF USINT;
	    usDecreaseActStepsActivated : USINT;
	    aDecreaseLimitsArrayEntry : ARRAY [0..ST151_MAXSTEPPING_MODES] OF USINT;
	  END_STRUCT;
#pragma pack(pop)
#pragma pack(push, 1)
	  t_s_ConfigModule1 : STRUCT
	    ChopperOffTime : UINT;
	    FastDecayTime : UINT;
	    FrequLimitRising64 : UDINT;
	    FrequLimitRising32 : UDINT;
	    FrequLimitRising16 : UDINT;
	    FrequLimitRising8 : UDINT;
	    FrequLimitRising4 : UDINT;
	    FrequLimitRising2 : UDINT;
	  END_STRUCT;
#pragma pack(pop)
#pragma pack(push, 1)
	  t_s_ConfigModule2 : STRUCT
	    HWRampdownDeltaFrequency : UINT;
	    HWRampdownDeltaTime : UINT;
	    IncrementalEncoderSettings : BSINT
	    [
	      1 ZeroPosInversion,
	      2 PhaseBInversion,
	      3 EdgeSampling1,
	      4 EdgeSampling2,
	      5 TTL_RS422Mode,
	      6 ABCountMode,
	      7 LatchType,
	      8 Bit8,
	    ];
	    BlankingTimeRegister : USINT;
	    reserved1 : USINT;
	    reserved2 : USINT;
	    RatedMaximumPowerWatt : UINT;
	    RegenResistance : UINT;
	    LoadThresholdWarning : USINT;
	    LoadThresholdDisableResistor : USINT;
	    MaximumCurrentReg : UINT;
	    ReducedCurrentReg : UINT;
	    LoadThresholdDisableBridge : USINT;
	  END_STRUCT;
#pragma pack(pop)
#pragma pack(push, 1)
	  t_s_ConfigModule3 : STRUCT
	    LatchCntZPuls : UINT;
	    LatchCntInput1Rising : UINT;
	    LatchCntInput1Falling : UINT;
	    LatchCntInput2Rising : UINT;
	    LatchCntInput2Falling : UINT;
	  END_STRUCT;
#pragma pack(pop)
#pragma pack(push, 1)
	  t_s_ConfigModule4 : STRUCT
	    ExtendedMotorStateReg1 : BINT
	    [
	      1 ZeroPosition,
	      2 OverTempWarning,
	      3 OverTempFailure,
	      4 OverCurrentFailureGND,
	      5 OverCurrentFailureBridge1,
	      6 OverCurrentFailureBridge2,
	      7 Encoder5VOk,
	      8 Bit8,
	      9 BridgeVoltageTooLow,
	      10 BridgeVoltageTooHigh,
	      11 ExternEnableSTO1,
	      12 ExternEnableSTO2,
	      13 SafetyStartUpOK,
	      14 MotorEnableError,
	      15 ThreeTimeSyncInLost,
	      16 SafeRampDownPending,
	    ];
	    ExtendedMotorStateReg2 : BSINT
	    [
	      1 LoadWarning,
	      2 LoadDisableBridge,
	      3 LoadDisableResistor,
	    ];
	    ActRegenResistorLoad : USINT;
	    u2tValue : UDINT;
	    HBridgeVoltage : INT;
	    HBridgeTemperature : INT;
	    CommutationCntHBridge1 : UINT;
	    CommutationCntHBridge2 : UINT;
	    OntimeCntHBridge1 : UINT;
	    OntimeCntHBridge2 : UINT;
	    bsControllerStateReg : BSINT
	    [
	      1 NoCalibData,
	      2 InvalidCalibData,
	      3 Bit3,
	      4 ControllerOP,
	      5 Bit5,
	      6 Bit6,
	      7 Bit7,
	      8 Bit8,
	    ];
	  END_STRUCT;
#pragma pack(pop)
#pragma pack(push, 1)
	  t_s_ConfigModule5 : STRUCT
	    bsControllerControlReg : BSINT
	    [
	      1 Bit1,
	      2 Bit2,
	      3 Bit3,
	      4 Bit4,
	      5 Bit5,
	      6 Bit6,
	      7 LoadConfigNew,
	      8 ControllerReset,
	    ];
	    reserved1 : UINT;
	    FrequLimitFalling32to64 : UDINT;
	    FrequLimitFalling16to32 : UDINT;
	    FrequLimitFalling8to16 : UDINT;
	    FrequLimitFalling4to8 : UDINT;
	    FrequLimitFalling2to4 : UDINT;
	    FrequLimitFalling1to2 : UDINT;
	    FastDecayTimeFallingStep : UINT;
	    ChopperOnTimeMin : UINT;
	  END_STRUCT;
#pragma pack(pop)
#pragma pack(push, 1)
	  t_s_ConfigModule6 : STRUCT
	    CurrentOffsetAdjBridge1 : INT;
	    CurrentOffsetAdjBridge2 : INT;
	  END_STRUCT;
#pragma pack(pop)
#pragma pack(push, 1)
	  t_s_ConfigModul : STRUCT
	    SDOData1 : t_s_ConfigModule1;
	    SDOData2 : t_s_ConfigModule2;
	    SDOData3 : t_s_ConfigModule3;
	    SDOData4 : t_s_ConfigModule4;
	    SDOData5 : t_s_ConfigModule5;
	    SDOData6 : t_s_ConfigModule6;
	  END_STRUCT;
#pragma pack(pop)
#pragma pack(push, 1)
	  t_SPI_CalibHeader : STRUCT
	    ud_Checksum : UDINT;
	    ud_ListVersion : UDINT;
	    ud_ListLength : UDINT;
	  END_STRUCT;
#pragma pack(pop)
#pragma pack(push, 1)
	  t_SPI_CalibData : STRUCT
	    SPI_Header : t_SPI_CalibHeader;
	    Offset0 : INT;
	    Multiplier0 : INT;
	    Divisor0 : UINT;
	    Offset1 : INT;
	    Multiplier1 : INT;
	    Divisor1 : UINT;
	    AI1Offset : INT;
	    AI1Multiplikator : INT;
	    AI1Divisor : INT;
	    AI2Offset : INT;
	    AI2Multiplikator : INT;
	    AI2Divisor : INT;
	    BridgeMaximumCurrent : UINT;
	    BridgeSupplyVoltageLowerThreshold : UINT;
	    BridgeSupplyVoltageUpperThreshold : UINT;
	    BridgeTemperatureWarningThreshold : UINT;
	    BridgeTemperatureErrorThreshold : UINT;
	  END_STRUCT;
#pragma pack(pop)
#pragma pack(push, 1)
	  t_SPIReadData : STRUCT
	    IDHeader : t_SPI_ListHeader;
	    udMaxDataLength : UDINT;
	    udActReadLength : UDINT;
	    udReadLength : UDINT;
	    udReadOffset : UDINT;
	  END_STRUCT;
#pragma pack(pop)
#pragma pack(push, 1)
	  t_SPIWriteData : STRUCT
	    usBytesToWrite : USINT;
	    usBytesActWrite : USINT;
	    usWriteOffset : USINT;
	  END_STRUCT;
#pragma pack(pop)
	END_TYPE
  //Servers:
	Online 	: SvrCh_DINT;
	EncoderPosition 	: SvrCh_DINT;
	ZPuls 	: SvrCh_DINT;
	ZPulsLatched 	: SvrCh_DINT;
	LatchPositionEncoderZeroPulse 	: SvrCh_DINT;
	LatchPositionInput1Rising 	: SvrCh_DINT;
	LatchPositionInput1Falling 	: SvrCh_DINT;
	LatchPositionInput2Rising 	: SvrCh_DINT;
	LatchPositionInput2Falling 	: SvrCh_DINT;
	Input1 	: SvrCh_DINT;
	Input1LatchedRising 	: SvrCh_DINT;
	Input1LatchedFalling 	: SvrCh_DINT;
	Input2 	: SvrCh_DINT;
	Input2LatchedRising 	: SvrCh_DINT;
	Input2LatchedFalling 	: SvrCh_DINT;
	Enable 	: SvrCh_DINT;
	ActPosition 	: SvrCh_DINT;
	SetFreqOut 	: SvrCh_DINT;
	TargetFreqOut 	: SvrCh_DINT;
	CurrentIncrease 	: SvrCh_DINT;
	ControlWord 	: SvrCh_DS402_Control;
	StateWord 	: SvrCh_DS402_State;
	ErrorInfo 	: SvrCh_BDINT;
	AxError 	: SvrCh_DINT;
	ErrorQuit 	: SvrCh_DINT;
	HWEnableSoftwareRampdown 	: SvrCh_DINT;
	HWRampdownDeltaFrequency 	: SvrCh_DINT;
	HWRampdownDeltaTime 	: SvrCh_DINT;
	MaxCurrent 	: SvrCh_DINT;
	CurrentOffsetAdjBridge1 	: SvrCh_DINT;
	CurrentOffsetAdjBridge2 	: SvrCh_DINT;
	ChopperOffTime 	: SvrCh_DINT;
	ChopperOnTimeMin 	: SvrCh_DINT;
	FastDecayTime 	: SvrCh_DINT;
	FastDecayTimeFallingStep 	: SvrCh_DINT;
	EnableSteps 	: SvrCh_bd_EnabledFreqLimit_PTofCls_ST151Base;
	FrequLimitIncrease2to1 	: SvrCh_UDINT;
	FrequLimitIncrease4to2 	: SvrCh_UDINT;
	FrequLimitIncrease8to4 	: SvrCh_UDINT;
	FrequLimitIncrease16to8 	: SvrCh_UDINT;
	FrequLimitIncrease32to16 	: SvrCh_UDINT;
	FrequLimitIncrease64to32 	: SvrCh_UDINT;
	FrequLimitDecrease1to2 	: SvrCh_UDINT;
	FrequLimitDecrease2to4 	: SvrCh_UDINT;
	FrequLimitDecrease4to8 	: SvrCh_UDINT;
	FrequLimitDecrease8to16 	: SvrCh_UDINT;
	FrequLimitDecrease16to32 	: SvrCh_UDINT;
	FrequLimitDecrease32to64 	: SvrCh_UDINT;
	RefreshValues 	: SvrCh_DINT;
	ExtendedStateWord 	: SvrCh_bd_ExtendedStateWord_PTofCls_ST151Base;
	HBridgeVoltage 	: SvrChCmd_DINT;
	HBridgeTemperature 	: SvrCh_DINT;
	ExternalEnable1 	: SvrCh_DINT;
	ExternalEnable2 	: SvrCh_DINT;
	ActRegenResistorLoad 	: SvrCh_DINT;
	VoltageOKEncoder 	: SvrCh_DINT;
  //Clients:
	InvertEncoder 	: CltCh_DINT;
	InvertZeroPosition 	: CltCh_DINT;
	EncoderSampling 	: CltCh_DINT;
	EncMode 	: CltCh_DINT;
	LatchType 	: CltCh_DINT;
	ABCountMode 	: CltCh_DINT;
	StallCurrentReduction 	: CltCh_DINT;
	StallCurrentWindow 	: CltCh_DINT;
	EnableRegenResistor 	: CltCh_DINT;
	RegenResistance 	: CltCh_DINT;
	RatedMaxPower 	: CltCh_DINT;
	LoadThresholdWarning 	: CltCh_DINT;
	LoadThresholdBridge 	: CltCh_DINT;
	LoadThresholdResistor 	: CltCh_DINT;
	SteppingHysteresis 	: CltCh_DINT;
	CompModeVST 	: CltCh_DINT;
	UseOszi 	: CltCh_DINT;
	toFreqLimitTable 	: CltCh_DINT;
  //Variables:
		sAccesses 	: t_Accesses;
		sAccessesOszi 	: t_AccessesOszi;
		eActStepping 	: e_ActStepMode;
		sWriteSDO 	: t_s_ConfigModul;
		sReadSDO 	: t_s_ConfigModul;
		udStallCurrentWindow 	: UDINT;
		uiPositionOld 	: UINT;
		eInitSSW 	: t_e_InitSSW;
		eInitSSWErrorStep 	: t_e_InitSSW;
		eResponseState 	: t_ResponseState;
		udSDOTimeOut 	: UDINT;
		aFrequencyLimit : ARRAY [0..ST151_MAXSTEPPING_MODES] OF t_FrequencyLimits;

		eActSDOConfigRdWr 	: t_e_SDOConfig;
		biReqSDOConfigRdWr 	: t_bi_ReqSDOConfig;
		bsRespSDOConfigRdWr 	: t_bi_ReqSDOConfig;
		usSDORetrys 	: USINT;
		uiOldCntVirtual 	: UINT;
		uiOldCntEncoder 	: UINT;
		sPLLRegister 	: t_PllRegister;
		sSPIReadData 	: t_SPIReadData;
		sSPIWriteData 	: t_SPIWriteData;
		sStepsNeeded 	: t_EnabledFreqLimit;
		dActDirection 	: DINT;
		dOldSetFrequ 	: DINT;
		udCyclicRefresh 	: UDINT;
		dFrequBandwith 	: DINT;
		dHighFrequencyLimit 	: DINT;
		sAdaptiveStepping 	: t_s_AdaptiveSteppingCalc;
		sLatchValues 	: t_LatchValues;
		udStartWaitTime 	: UDINT;
		udLimitsHysteresis 	: UDINT;
		usCompModeVST 	: USINT;
  //Functions:
				//! <Function Comment="Init-Methode of Class.&#13;&#10;&#13;&#10;This Methode needs to get called. In case the Methode gets overwritten, a call needs to bet installed." Name="Init"/>
	FUNCTION VIRTUAL GLOBAL Init;

	FUNCTION ST151Base
		VAR_OUTPUT
			ret_code 	: ConfStates;
		END_VAR;
				//! <Function Comment="Realtime Update Methode which runs in PreScan." Name="UpdateRt"/>
	FUNCTION VIRTUAL GLOBAL UpdateRt;
				//! <Function Comment="Realtime Update Methode which runs in PostScan." Name="UpdateRtPostScan"/>
	FUNCTION VIRTUAL GLOBAL UpdateRtPostScan;
				//! <Function Comment="Cyclic Update Methode which runs in PostScan." Name="UpdateCy"/>
	FUNCTION VIRTUAL GLOBAL UpdateCy;

	FUNCTION VIRTUAL GLOBAL AddAccesses
		VAR_OUTPUT
			eModuleInitState 	: iprStates;
		END_VAR;
				//! <Function Comment="Methode is called if this Module gets connected." Name="ConnectEvent"/>
	FUNCTION VIRTUAL GLOBAL ConnectEvent;
				//! <Function Comment="Methode is called if this Module gets disconnected." Name="DisconnectEvent"/>
	FUNCTION VIRTUAL GLOBAL DisconnectEvent;
				//! <Function Comment="Methode should be used to run a Statemachine to Initialize the Module." Name="InitModule"/>
	FUNCTION VIRTUAL GLOBAL InitModule
		VAR_OUTPUT
			eModuleInitState 	: iprStates;			//! <Variable Comment="Return BUSY until the Initialisation is finished." Name="InitModule.eModuleInitState"/>
		END_VAR;
				//! <Function Comment="This Methode should be used, to check the DeviceID of the Module." Name="CheckDeviceID"/>
	FUNCTION VIRTUAL GLOBAL CheckDeviceID
		VAR_INPUT
			udID2Check 	: UDINT;			//! <Variable Comment="Device ID of connected Module." Name="CheckDeviceID.udID2Check"/>
		END_VAR
		VAR_OUTPUT
			bIsOK 	: BOOL;			//! <Variable Comment="FALSE = Wrong DeviceID for Module&#13;&#10;TRUE  = DeviceID of Module is correct" Name="CheckDeviceID.bIsOK"/>
		END_VAR;
				//! <Function Comment="Methode to receive the Response in case of SDO-Communication." Name="ReceiveSDOResponse"/>
	FUNCTION VIRTUAL ReceiveSDOResponse
		VAR_INPUT
			eCommand 	: t_SDIAS_SDO_Cmd;			//! <Variable Comment="Type of SDO-Command" Name="ReceiveSDOResponse.eCommand"/>
			hOffset 	: HINT;			//! <Variable Comment="Address-Offset in Module." Name="ReceiveSDOResponse.hOffset"/>
			usLength 	: USINT;			//! <Variable Comment="Length of Data." Name="ReceiveSDOResponse.usLength"/>
			eResult 	: iprStates;			//! <Variable Comment="State of SDO-Communication." Name="ReceiveSDOResponse.eResult"/>
			pResponseBuffer 	: ^USINT;			//! <Variable Comment="Pointer of ResponseBuffer, where the SDO-Data is located." Name="ReceiveSDOResponse.pResponseBuffer"/>
			ResponseLength 	: USINT;			//! <Variable Comment="Size of the ResponseBuffer." Name="ReceiveSDOResponse.ResponseLength"/>
		END_VAR
		VAR_OUTPUT
			ret_code 	: iprStates;			//! <Variable Comment="Indicates if the Methode was successful." Name="ReceiveSDOResponse.ret_code"/>
		END_VAR;

	FUNCTION VIRTUAL GetTaskCfg
		VAR_OUTPUT
			TaskCfg 	: BDINT;			//! <Variable Comment="Select which tasks will be available for this module:&#13;&#10;Bit0..Realtime PreScan&#13;&#10;Bit1..Realtime PostScan&#13;&#10;Bit2..Cyclic&#13;&#10;&#13;&#10;e.g. if only realtime postscan is needed:&#13;&#10;2#010" Name="GetTaskCfg.TaskCfg"/>
		END_VAR;

	FUNCTION VIRTUAL GLOBAL GetDeviceID
		VAR_OUTPUT
			output 	: UDINT;
		END_VAR;

	FUNCTION CalcAdaptiveMicroStepping
		VAR_INPUT
			dTargetFrequency 	: DINT;
			dActSetFrequency 	: DINT;
		END_VAR
		VAR_OUTPUT
			dRetCode 	: DINT;
		END_VAR;

	FUNCTION SDORdWrData
		VAR_OUTPUT
			dRetCode 	: iprStates;
		END_VAR;

	FUNCTION CalcSimpleMode;
				//! <Function Comment="Start measuring of h-bridge voltage." Name="StartMeasure"/>
	FUNCTION GLOBAL StartMeasure
		VAR_INPUT
			pData 	: ^void;			//! <Variable Comment="pointer to memory area which must have a minimum size of 1024 bytes." Name="StartMeasure.pData"/>
			uiTriggerLevel 	: UINT;			//! <Variable Comment="set the trigger level in xx.xx [V]." Name="StartMeasure.uiTriggerLevel"/>
			uiSamplePrescaler 	: UINT;			//! <Variable Comment="Set a prescaler for recording of values.&#13;&#10;The values are recorded at 62,5 intervals.&#13;&#10;1 .. every value is recorded.&#13;&#10;10 .. every tenth value is recorded." Name="StartMeasure.uiSamplePrescaler"/>
			bStartStopMeasure 	: BOOL;			//! <Variable Comment="Start or stop measuring.&#13;&#10;0 .. stop measure&#13;&#10;1 .. start measure" Name="StartMeasure.bStartStopMeasure"/>
			usTriggerSetting 	: USINT;			//! <Variable Comment="set trigger mode:&#13;&#10;0 .. rising edge&#13;&#10;1 .. falling edge&#13;&#10;2 .. forced trigger" Name="StartMeasure.usTriggerSetting"/>
			usTriggerOffset 	: USINT;			//! <Variable Comment="set offset for trigger record:&#13;&#10;0 .. 0%&#13;&#10;1 .. -25%&#13;&#10;2 .. -50%&#13;&#10;3 .. -75%" Name="StartMeasure.usTriggerOffset"/>
		END_VAR
		VAR_OUTPUT
			dRetCode 	: DINT;			//! <Variable Comment="Returnvalue of function.&#13;&#10;0 .. ok&#13;&#10;-1 .. function not activated (client &quot;UseOszi&quot;)&#13;&#10;-2 .. data pointer not valid&#13;&#10;-3 .. usTriggerSetting not valid&#13;&#10;-4 .. usTriggerOffset not valid&#13;&#10;-5 .. measure is already started" Name="StartMeasure.dRetCode"/>
		END_VAR;

	FUNCTION GetMeasureData
		VAR_INPUT
			pData 	: ^void;
		END_VAR;

	FUNCTION SetSDORdWrStep
		VAR_INPUT
			eActStep 	: t_e_SDOConfig;
		END_VAR
		VAR_OUTPUT
			eNextStep 	: t_e_SDOConfig;
		END_VAR;
				//! <Function Comment="Get state of measuring." Name="GetMeasureState"/>
	FUNCTION GLOBAL GetMeasureState
		VAR_INPUT
			pbTriggered 	: ^BOOL := NIL;			//! <Variable Comment="Pointer to bool value.&#13;&#10;0 .. not triggerd&#13;&#10;1 .. triggerd" Name="GetMeasureState.pbTriggered"/>
		END_VAR
		VAR_OUTPUT
			dRetCode 	: DINT;			//! <Variable Comment="Returnvalue of methode.&#13;&#10;0 .. measure ready&#13;&#10;1 .. measure busy&#13;&#10;&#13;&#10;-1 .. pointer for pbTriggerd is not valid.&#13;&#10;-2 .. pointer for pbBufferOverflow is not valid.&#13;&#10;-3 .. no measure started&#13;&#10;" Name="GetMeasureState.dRetCode"/>
		END_VAR;

	FUNCTION GLOBAL GetActFreqLimits
		VAR_INPUT
			usValueIncDec 	: USINT;
			usArrayEntry 	: USINT;
			pusActCompMode 	: ^USINT;
		END_VAR
		VAR_OUTPUT
			udData 	: UDINT;
		END_VAR;

	FUNCTION VIRTUAL GLOBAL ZPulsLatched::Read
		VAR_OUTPUT
			output (EAX) 	: DINT;
		END_VAR;

	FUNCTION VIRTUAL GLOBAL Input1LatchedRising::Read
		VAR_OUTPUT
			output (EAX) 	: DINT;
		END_VAR;

	FUNCTION VIRTUAL GLOBAL Input1LatchedFalling::Read
		VAR_OUTPUT
			output (EAX) 	: DINT;
		END_VAR;

	FUNCTION VIRTUAL GLOBAL Input2LatchedRising::Read
		VAR_OUTPUT
			output (EAX) 	: DINT;
		END_VAR;

	FUNCTION VIRTUAL GLOBAL Input2LatchedFalling::Read
		VAR_OUTPUT
			output (EAX) 	: DINT;
		END_VAR;

	FUNCTION VIRTUAL GLOBAL Enable::Write
		VAR_INPUT
			input (EAX) 	: DINT;
		END_VAR
		VAR_OUTPUT
			result (EAX) 	: DINT;
		END_VAR;

	FUNCTION VIRTUAL GLOBAL SetFreqOut::Write
		VAR_INPUT
			input (EAX) 	: DINT;
		END_VAR
		VAR_OUTPUT
			result (EAX) 	: DINT;
		END_VAR;

	FUNCTION VIRTUAL GLOBAL TargetFreqOut::Write
		VAR_INPUT
			input (EAX) 	: DINT;
		END_VAR
		VAR_OUTPUT
			result (EAX) 	: DINT;
		END_VAR;

	FUNCTION VIRTUAL GLOBAL CurrentIncrease::Write
		VAR_INPUT
			input (EAX) 	: DINT;
		END_VAR
		VAR_OUTPUT
			result (EAX) 	: DINT;
		END_VAR;

	FUNCTION VIRTUAL GLOBAL ControlWord::Write
		VAR_INPUT
			input (EAX) 	: DS402_Control;
		END_VAR
		VAR_OUTPUT
			result (EAX) 	: DS402_Control;
		END_VAR;

	FUNCTION VIRTUAL GLOBAL ErrorQuit::Write
		VAR_INPUT
			input (EAX) 	: DINT;
		END_VAR
		VAR_OUTPUT
			result (EAX) 	: DINT;
		END_VAR;

	FUNCTION VIRTUAL GLOBAL HWEnableSoftwareRampdown::Write
		VAR_INPUT
			input (EAX) 	: DINT;
		END_VAR
		VAR_OUTPUT
			result (EAX) 	: DINT;
		END_VAR;

	FUNCTION VIRTUAL GLOBAL HWRampdownDeltaFrequency::Write
		VAR_INPUT
			input (EAX) 	: DINT;
		END_VAR
		VAR_OUTPUT
			result (EAX) 	: DINT;
		END_VAR;

	FUNCTION VIRTUAL GLOBAL HWRampdownDeltaTime::Write
		VAR_INPUT
			input (EAX) 	: DINT;
		END_VAR
		VAR_OUTPUT
			result (EAX) 	: DINT;
		END_VAR;

	FUNCTION VIRTUAL GLOBAL MaxCurrent::Write
		VAR_INPUT
			input (EAX) 	: DINT;
		END_VAR
		VAR_OUTPUT
			result (EAX) 	: DINT;
		END_VAR;

	FUNCTION VIRTUAL GLOBAL CurrentOffsetAdjBridge1::Write
		VAR_INPUT
			input (EAX) 	: DINT;
		END_VAR
		VAR_OUTPUT
			result (EAX) 	: DINT;
		END_VAR;

	FUNCTION VIRTUAL GLOBAL CurrentOffsetAdjBridge2::Write
		VAR_INPUT
			input (EAX) 	: DINT;
		END_VAR
		VAR_OUTPUT
			result (EAX) 	: DINT;
		END_VAR;
				//! <Function Comment="Set fixed off-time of the PWM  [20ns steps] as init value.&#13;&#10;Valid range is from 1500 up to 65535." Name="ChopperOffTime.Write"/>
	FUNCTION VIRTUAL GLOBAL ChopperOffTime::Write
		VAR_INPUT
			input (EAX) 	: DINT;
		END_VAR
		VAR_OUTPUT
			result (EAX) 	: DINT;
		END_VAR;

	FUNCTION VIRTUAL GLOBAL ChopperOnTimeMin::Write
		VAR_INPUT
			input (EAX) 	: DINT;
		END_VAR
		VAR_OUTPUT
			result (EAX) 	: DINT;
		END_VAR;

	FUNCTION VIRTUAL GLOBAL FastDecayTime::Write
		VAR_INPUT
			input (EAX) 	: DINT;
		END_VAR
		VAR_OUTPUT
			result (EAX) 	: DINT;
		END_VAR;

	FUNCTION VIRTUAL GLOBAL FastDecayTimeFallingStep::Write
		VAR_INPUT
			input (EAX) 	: DINT;
		END_VAR
		VAR_OUTPUT
			result (EAX) 	: DINT;
		END_VAR;

	FUNCTION VIRTUAL GLOBAL EnableSteps::Write
		VAR_INPUT
			input (EAX) 	: ST151Base::bd_EnabledFreqLimit;
		END_VAR
		VAR_OUTPUT
			result (EAX) 	: ST151Base::bd_EnabledFreqLimit;
		END_VAR;

	FUNCTION VIRTUAL GLOBAL FrequLimitIncrease2to1::Write
		VAR_INPUT
			input (EAX) 	: UDINT;
		END_VAR
		VAR_OUTPUT
			result (EAX) 	: UDINT;
		END_VAR;

	FUNCTION VIRTUAL GLOBAL FrequLimitIncrease4to2::Write
		VAR_INPUT
			input (EAX) 	: UDINT;
		END_VAR
		VAR_OUTPUT
			result (EAX) 	: UDINT;
		END_VAR;

	FUNCTION VIRTUAL GLOBAL FrequLimitIncrease8to4::Write
		VAR_INPUT
			input (EAX) 	: UDINT;
		END_VAR
		VAR_OUTPUT
			result (EAX) 	: UDINT;
		END_VAR;

	FUNCTION VIRTUAL GLOBAL FrequLimitIncrease16to8::Write
		VAR_INPUT
			input (EAX) 	: UDINT;
		END_VAR
		VAR_OUTPUT
			result (EAX) 	: UDINT;
		END_VAR;

	FUNCTION VIRTUAL GLOBAL FrequLimitIncrease32to16::Write
		VAR_INPUT
			input (EAX) 	: UDINT;
		END_VAR
		VAR_OUTPUT
			result (EAX) 	: UDINT;
		END_VAR;

	FUNCTION VIRTUAL GLOBAL FrequLimitIncrease64to32::Write
		VAR_INPUT
			input (EAX) 	: UDINT;
		END_VAR
		VAR_OUTPUT
			result (EAX) 	: UDINT;
		END_VAR;

	FUNCTION VIRTUAL GLOBAL FrequLimitDecrease1to2::Write
		VAR_INPUT
			input (EAX) 	: UDINT;
		END_VAR
		VAR_OUTPUT
			result (EAX) 	: UDINT;
		END_VAR;

	FUNCTION VIRTUAL GLOBAL FrequLimitDecrease2to4::Write
		VAR_INPUT
			input (EAX) 	: UDINT;
		END_VAR
		VAR_OUTPUT
			result (EAX) 	: UDINT;
		END_VAR;

	FUNCTION VIRTUAL GLOBAL FrequLimitDecrease4to8::Write
		VAR_INPUT
			input (EAX) 	: UDINT;
		END_VAR
		VAR_OUTPUT
			result (EAX) 	: UDINT;
		END_VAR;

	FUNCTION VIRTUAL GLOBAL FrequLimitDecrease8to16::Write
		VAR_INPUT
			input (EAX) 	: UDINT;
		END_VAR
		VAR_OUTPUT
			result (EAX) 	: UDINT;
		END_VAR;

	FUNCTION VIRTUAL GLOBAL FrequLimitDecrease16to32::Write
		VAR_INPUT
			input (EAX) 	: UDINT;
		END_VAR
		VAR_OUTPUT
			result (EAX) 	: UDINT;
		END_VAR;

	FUNCTION VIRTUAL GLOBAL FrequLimitDecrease32to64::Write
		VAR_INPUT
			input (EAX) 	: UDINT;
		END_VAR
		VAR_OUTPUT
			result (EAX) 	: UDINT;
		END_VAR;

	FUNCTION VIRTUAL GLOBAL RefreshValues::Write
		VAR_INPUT
			input (EAX) 	: DINT;
		END_VAR
		VAR_OUTPUT
			result (EAX) 	: DINT;
		END_VAR;
  //Tables:
	FUNCTION @STD
		VAR_OUTPUT
			ret_code	: CONFSTATES;
		END_VAR;
	FUNCTION GLOBAL TAB @CT_;
END_CLASS;

FUNCTION VIRTUAL GLOBAL ST151Base::Init
  //call base class
  SdiasBase::Init();

  if _FirstScan then
    //initialize CompModeVST to avoid division error if hardware is not ok
    usCompModeVST := 1;

    // show deactivated at startup (was init value on server before, but since it has not been written to the module on startup it's a init value here now)
    TargetFreqOut := -1;
  end_if;

END_FUNCTION

FUNCTION VIRTUAL GLOBAL ST151Base::UpdateRt
  VAR
    ui_temp       : UINT;
    si_delta      : INT;
    TempReadData  : t_s_ReadData;
    bsLatchActual : t_bs_IsyncValue;
    TempReadOsziData : t_s_OsziRead;
    usTempCnt : USINT;
    uiActReadLength : UINT;
    uiTempLength : UINT;
    uiToLastEntryLength : UINT;
    bTempBool : BOOL;
    tmpStateWord : DS402_State;
  END_VAR

  TempReadData := sAccesses.pReadData^;

  ZPuls := TempReadData.StateWord.LatchIncZero;

  if TempReadData.StateWord.LatchIncZero = 1 then
    ZPulsLatched := TempReadData.StateWord.LatchIncZero;
  end_if;

  //Update Digital Inputs
  Input1 := TempReadData.StateWord.DigIn1;
  Input2 := TempReadData.StateWord.DigIn2;

  bsLatchActual := ((TempReadData.StateWord shr 9) AND 2#11111)$t_bs_IsyncValue;

  if EncoderSampling & LatchType then
    if bsLatchActual.IncZero then
      sLatchValues.uiISyncIncZeroOldCounter  := uiOldCntEncoder;
      sLatchValues.sdISyncIncZeroOldPosition := EncoderPosition;
    end_if;
    if bsLatchActual.DigIn1Rise then
      sLatchValues.uiISyncDigIn1RiseOldCounter  := uiOldCntEncoder;
      sLatchValues.sdISyncDigIn1RiseOldPosition := EncoderPosition;
    end_if;
    if bsLatchActual.DigIn1Fall then
      sLatchValues.uiISyncDigIn1FallOldCounter  := uiOldCntEncoder;
      sLatchValues.sdISyncDigIn1FallOldPosition := EncoderPosition;
    end_if;
    if bsLatchActual.DigIn2Rise then
      sLatchValues.uiISyncDigIn2RiseOldCounter  := uiOldCntEncoder;
      sLatchValues.sdISyncDigIn2RiseOldPosition := EncoderPosition;
    end_if;
    if bsLatchActual.DigIn2Fall then
      sLatchValues.uiISyncDigIn2FallOldCounter  := uiOldCntEncoder;
      sLatchValues.sdISyncDigIn2FallOldPosition := EncoderPosition;
    end_if;
  else
    //virtual position have no z puls
    if bsLatchActual.IncZero then
      sLatchValues.uiISyncIncZeroOldCounter  := uiOldCntEncoder;
      sLatchValues.sdISyncIncZeroOldPosition := EncoderPosition;
    end_if;
    if bsLatchActual.DigIn1Rise then
      sLatchValues.uiISyncDigIn1RiseOldCounter  := uiOldCntVirtual;
      sLatchValues.sdISyncDigIn1RiseOldPosition := ActPosition;
    end_if;
    if bsLatchActual.DigIn1Fall then
      sLatchValues.uiISyncDigIn1FallOldCounter  := uiOldCntVirtual;
      sLatchValues.sdISyncDigIn1FallOldPosition := ActPosition;
    end_if;
    if bsLatchActual.DigIn2Rise then
      sLatchValues.uiISyncDigIn2RiseOldCounter  := uiOldCntVirtual;
      sLatchValues.sdISyncDigIn2RiseOldPosition := ActPosition;
    end_if;
    if bsLatchActual.DigIn2Fall then
      sLatchValues.uiISyncDigIn2FallOldCounter  := uiOldCntVirtual;
      sLatchValues.sdISyncDigIn2FallOldPosition := ActPosition;
    end_if;
  end_if;

  //actual encoder position
  ui_temp         := TempReadData.IncrementalEncoderValue;
  si_delta        := to_int(ui_temp - uiOldCntEncoder);
  EncoderPosition += to_dint(si_delta);
  uiOldCntEncoder := ui_temp;

  //actual virtual position
  ui_temp         := TempReadData.ActPos;
  si_delta        := to_int(ui_temp - uiOldCntVirtual);
  ActPosition     += to_dint(si_delta/usCompModeVST);
  uiOldCntVirtual := ui_temp;
  if si_delta mod usCompModeVST then
    if si_delta > 0 then
      uiOldCntVirtual -= 1;
    else
      uiOldCntVirtual += 1;
    end_if;
  end_if;

  //check for changed latched bits while reading latch counter
  if sLatchValues.bResetActiveSyncValue
  & bsLatchActual <> sLatchValues.bsValidISyncValue then
    sLatchValues.bsActiveISyncValue    := 0;
    sLatchValues.bResetActiveSyncValue := FALSE;
  end_if;

  // check for latched bits
  if bsLatchActual | sLatchValues.bsLatchReaded then

    //Input1 rising latched
    if ( TempReadData.StateWord.LatchDigIn1Rise ) | sLatchValues.bsLatchReaded.DigIn1Rise then
      sLatchValues.bsLatchReaded.DigIn1Rise := FALSE;
      Input1LatchedRising      := TempReadData.StateWord.LatchDigIn1Rise; //Reset of Bit is done with Read-Access
    end_if;

    //Input1 falling latched
    if ( TempReadData.StateWord.LatchDigIn1Fall ) | sLatchValues.bsLatchReaded.DigIn1Fall then
      sLatchValues.bsLatchReaded.DigIn1Fall := FALSE;
      Input1LatchedFalling     := TempReadData.StateWord.LatchDigIn1Fall; //Reset of Bit is done with Read-Access
    end_if;

    //Input2 rising latched
    if ( TempReadData.StateWord.LatchDigIn2Rise ) | sLatchValues.bsLatchReaded.DigIn2Rise then
      sLatchValues.bsLatchReaded.DigIn2Rise := FALSE;
      Input2LatchedRising      := TempReadData.StateWord.LatchDigIn2Rise; //Reset of Bit is done with Read-Access
    end_if;

    //Input2 falling latched
    if ( TempReadData.StateWord.LatchDigIn2Fall ) | sLatchValues.bsLatchReaded.DigIn2Fall then
      sLatchValues.bsLatchReaded.DigIn2Fall := FALSE;
      Input2LatchedFalling     := TempReadData.StateWord.LatchDigIn2Fall; //Reset of Bit is done with Read-Access
    end_if;

    //Zpuls Latched
    if sLatchValues.bsLatchReaded.IncZero then
      sLatchValues.bsLatchReaded.IncZero := FALSE;
      ZPulsLatched          := TempReadData.StateWord.LatchIncZero;
    end_if;

    if bsLatchActual <> sLatchValues.bsActiveISyncValue then
      //save actual latch values to read per sdo.
      sLatchValues.bsActiveISyncValue    := sLatchValues.bsActiveISyncValue or bsLatchActual;
    end_if;
  end_if;

  tmpStateWord                    := 0;
  tmpStateWord.OperationEnabled   := TempReadData.StateWord.MotorEnabled;
  tmpStateWord.ReadyToSwitchOn    := TempReadData.StateWord.ReadyToSwitchOn;
  bTempBool                       := TempReadData.StateWord.ReadyToSwitchOn AND (TempReadData.StateWord.STOSwitchOff = 0);
  tmpStateWord.SwitchedOn         := bTempBool AND (TempReadData.StateWord.Fault = 0);
  tmpStateWord.Warning            := ( TempReadData.StateWord.TemperatureOK = 0 );
  AxError := tmpStateWord.Fault   := TempReadData.StateWord.Fault;
  ErrorInfo$BINT                  := (TempReadData.StateWord and ST151_ERROR_BITMASK_STATE_WORD) xor 0x0004;
  StateWord                       := tmpStateWord;
  //class is ok
  Online  := 1;

  //read oszi data if activated
  if UseOszi then
    TempReadOsziData := sAccessesOszi.pReadHeader^;
    uiActReadLength  := 0;
    case sAccessesOszi.eOsziData of
      //*********************************************************************************************************
      _OsziDataIdle:

      //*********************************************************************************************************
      _OsziTriggerStart:
        sAccessesOszi.eOsziData := _OsziResetTrigger;

      //*********************************************************************************************************
      _OsziResetTrigger:
        sAccessesOszi.sWriteOszi.ControlOszi.StartTriggering := FALSE;
        udStartWaitTime := ops.tAbsolute;
//        sAccessesOszi.eOsziData := _OsziWait4Reset;

      //*********************************************************************************************************
      _OsziWait4Reset:
        if (ops.tAbsolute-udStartWaitTime) >= 5 then
          sAccessesOszi.eOsziData := _OsziWait4Trigger;
        end_if;

      //*********************************************************************************************************
      _OsziWait4Trigger:
        sAccessesOszi.sLastOsziState.StateOszi := TempReadOsziData.StateOszi;
        if TempReadOsziData.StateOszi.Ready & TempReadOsziData.StateOszi.Triggered then
          sAccessesOszi.sLastOsziState       := TempReadOsziData;
          //enable accesses
          for usTempCnt := 0 to ST151_OSZI_MAX_PDOREAD-1 do
            if sAccessesOszi.aReadDataControl[usTempCnt].pControlByte then
              //Start Read-Access to Module (Set ControlWord in DPRam)
              sAccessesOszi.aReadDataControl[usTempCnt].pControlByte^ := TRUE;
              uiActReadLength += ST151_OSZI_ONE_PDOSIZE;
            end_if;
          end_for;
          sAccessesOszi.eOsziData := _OsziDisableRead;
        end_if;

      //*********************************************************************************************************
      _OsziDisableRead:
        //disable read access
        for usTempCnt := 0 to ST151_OSZI_MAX_PDOREAD-1 do
          if sAccessesOszi.aReadDataControl[usTempCnt].pControlByte then
            //Stop Read-Access to Module (Set ControlWord in DPRam)
            sAccessesOszi.aReadDataControl[usTempCnt].pControlByte^ := FALSE;
            uiActReadLength += ST151_OSZI_ONE_PDOSIZE;
          end_if;
        end_for;
        sAccessesOszi.eOsziData := _OsziWait4Data;

      //*********************************************************************************************************
      _OsziWait4Data:
        sAccessesOszi.eOsziData := _OsziGetData;

      //*********************************************************************************************************
      _OsziGetData:
        for usTempCnt := 0 to ST151_OSZI_MAX_PDOREAD-1 do
          uiTempLength := (usTempCnt+1)*ST151_OSZI_ONE_PDOSIZE;
          if uiTempLength > ST151_OSZI_BUFFER_SIZE then
            uiTempLength := ST151_OSZI_BUFFER_SIZE - (usTempCnt*ST151_OSZI_ONE_PDOSIZE);
          else
            uiTempLength := ST151_OSZI_ONE_PDOSIZE;
          end_if;
          _memcpy(ptr1:=#sAccessesOszi.aLastOsziData[(((ST151_OSZI_ONE_PDOSIZE*usTempCnt)/sizeof(UINT)))], ptr2:=sAccessesOszi.apOsziData[usTempCnt], cntr:=uiTempLength);
        end_for;

        uiToLastEntryLength := (sAccessesOszi.sLastOsziState.PointerOnLastSampleData$UINT - ST151_OSZI_READPOINTER_OFFSET + sizeof(UINT));
        sAccessesOszi.pLastEntryOsziData := (#sAccessesOszi.aLastOsziData[0] + uiToLastEntryLength - sizeof(UINT));
        sAccessesOszi.uiDatalength1      := uiToLastEntryLength;

        if uiToLastEntryLength = ST151_OSZI_BUFFER_SIZE then
          sAccessesOszi.pFirstEntryOsziData := #sAccessesOszi.aLastOsziData[0];
          sAccessesOszi.bSplitBuffer        := FALSE;
        else
          sAccessesOszi.uiDatalength2       := ST151_OSZI_BUFFER_SIZE-sAccessesOszi.uiDatalength1;
          sAccessesOszi.pFirstEntryOsziData := (#sAccessesOszi.aLastOsziData+(ST151_OSZI_BUFFER_SIZE-sAccessesOszi.uiDatalength2));
          sAccessesOszi.bSplitBuffer        := TRUE;
        end_if;

        //copy data to application
        GetMeasureData(pData:=sAccessesOszi.pToExternData);
        sAccessesOszi.bDataReady := TRUE;
        sAccessesOszi.eOsziData  := _OsziFinished;

      //*********************************************************************************************************
      _OsziFinished:
        sAccessesOszi.eOsziData  := _OsziDataIdle;

    end_case;
  end_if;

END_FUNCTION

FUNCTION VIRTUAL GLOBAL ST151Base::UpdateRtPostScan

  sAccesses.sWriteData.ControlWord.HWEnableSofwareRampdownToggleBit := sAccesses.sWriteData.ControlWord.HWEnableSofwareRampdownToggleBit XOR to_BOOL(HWEnableSoftwareRampdown);
  sAccesses.pWriteData^ := sAccesses.sWriteData;

  if sAccesses.sWriteData.ControlWord.FaultReset then
    sAccesses.sWriteData.ControlWord.FaultReset := FALSE;
    sAccesses.sWriteData.ControlWord.QuitSTOOff := FALSE;
    sAccesses.sWriteData.ControlWord.RegenResistorFaultReset := FALSE;
    ControlWord.ResetFault := FALSE;
    ErrorQuit              := 0;
  end_if;

  if UseOszi then
    sAccessesOszi.pWriteHeader^ := sAccessesOszi.sWriteOszi;
    if sAccessesOszi.eOsziData = _OsziResetTrigger then
      if sAccessesOszi.sWriteOszi.ControlOszi.CancelTrigger = FALSE then
        sAccessesOszi.eOsziData := _OsziWait4Reset;
      else
        sAccessesOszi.eOsziData := _OsziFinished;
      end_if;
      sAccessesOszi.sWriteOszi.ControlOszi.StartTriggering := FALSE;
      sAccessesOszi.sWriteOszi.ControlOszi.CancelTrigger := FALSE;
    end_if;
  end_if;

END_FUNCTION

FUNCTION VIRTUAL GLOBAL ST151Base::UpdateCy
  VAR
  	dRetCode : iprStates;
    iDeltaPos : INT;
    pbiTempErrorInfo :^BINT;
    usTempCompMode : USINT;
  END_VAR

  //Refresh cyclic values
  if (((ops.tAbsolute - udCyclicRefresh) >= ST151_CYCLICREFRESHDATA_TIME) & (RefreshValues = 1)) then
    udCyclicRefresh := ops.tAbsolute;
    biReqSDOConfigRdWr.ReadConfigSDO4 := TRUE;
  end_if;

  if (sLatchValues.bsActiveISyncValue & sLatchValues.bResetActiveSyncValue = FALSE) then
    biReqSDOConfigRdWr.ReadConfigSDO3 := TRUE;
  end_if;

  //read-write sdo data to module
  if biReqSDOConfigRdWr | eActSDOConfigRdWr <> _SDOConfig_Idle then
    dRetCode := SDORdWrData();
    if dRetCode = Ready then
      //all OK
    elsif dRetCode = Error then
      //error occured while read - write sdo
    end_if;
  end_if;

  //new cyclic data is available
  if bsRespSDOConfigRdWr.ReadConfigSDO4 = TRUE then
    if RefreshValues <> 0 then
      ExtendedStateWord    := sReadSDO.SDOData4.ExtendedMotorStateReg1$bd_ExtendedStateWord and 0xFFFFFF;
  //    DC24VOk := sReadSDO.SDOData3.ExtendedMotorStateReg1.Bit8;
      VoltageOKEncoder     := sReadSDO.SDOData4.ExtendedMotorStateReg1.Encoder5VOk;
      HBridgeVoltage       := sReadSDO.SDOData4.HBridgeVoltage;
      HBridgeTemperature   := sReadSDO.SDOData4.HBridgeTemperature;
      ExternalEnable1      := sReadSDO.SDOData4.ExtendedMotorStateReg1.ExternEnableSTO1;
      ExternalEnable2      := sReadSDO.SDOData4.ExtendedMotorStateReg1.ExternEnableSTO2;
      ActRegenResistorLoad  := sReadSDO.SDOData4.ActRegenResistorLoad;
      pbiTempErrorInfo     := (#ErrorInfo+2)$^BINT;
      pbiTempErrorInfo^    := (sReadSDO.SDOData4.ExtendedMotorStateReg1 and ST151_ERROR_BITMASK_EXTENDED_STATE_WORD) xor 0x1C00;
      pbiTempErrorInfo^.1  := sReadSDO.SDOData4.ExtendedMotorStateReg2.LoadWarning;
      pbiTempErrorInfo^.7  := sReadSDO.SDOData4.ExtendedMotorStateReg2.LoadDisableBridge;
      pbiTempErrorInfo^.8  := sReadSDO.SDOData4.ExtendedMotorStateReg2.LoadDisableResistor;
      if RefreshValues = 2 then
        RefreshValues := 0;
      end_if;
    end_if;;
    bsRespSDOConfigRdWr.ReadConfigSDO4 := FALSE;
  end_if;

  //new latchposition is available
  if bsRespSDOConfigRdWr.ReadConfigSDO3 = TRUE then
    if sLatchValues.bsValidISyncValue then
      if LatchType = 1 then
        usTempCompMode := 1;
      else
        usTempCompMode := usCompModeVST;
      end_if;
        if sLatchValues.bsValidISyncValue.IncZero then
          sLatchValues.uiLatchInputZero := sReadSDO.SDOData3.LatchCntZPuls;
          iDeltaPos := to_int(sLatchValues.uiLatchInputZero - sLatchValues.uiISyncIncZeroOldCounter);
          LatchPositionEncoderZeroPulse := sLatchValues.sdISyncIncZeroOldPosition + to_dint(iDeltaPos);
        end_if;
        if sLatchValues.bsValidISyncValue.DigIn1Rise & sReadSDO.SDOData3.LatchCntInput1Rising then
          sLatchValues.uiLatchInputDigIn1Rising := sReadSDO.SDOData3.LatchCntInput1Rising;
          iDeltaPos := to_int(sLatchValues.uiLatchInputDigIn1Rising - sLatchValues.uiISyncDigIn1RiseOldCounter)/usTempCompMode;
          LatchPositionInput1Rising := sLatchValues.sdISyncDigIn1RiseOldPosition + to_dint(iDeltaPos);
        end_if;
        if sLatchValues.bsValidISyncValue.DigIn1Fall & sReadSDO.SDOData3.LatchCntInput1Falling then
          sLatchValues.uiLatchInputDigIn1Falling := sReadSDO.SDOData3.LatchCntInput1Falling;
          iDeltaPos := to_int(sLatchValues.uiLatchInputDigIn1Falling - sLatchValues.uiISyncDigIn1FallOldCounter)/usTempCompMode;
          LatchPositionInput1Falling := sLatchValues.sdISyncDigIn1FallOldPosition + to_dint(iDeltaPos);
        end_if;
        if sLatchValues.bsValidISyncValue.DigIn2Rise  & sReadSDO.SDOData3.LatchCntInput2Rising then
          sLatchValues.uiLatchInputDigIn2Rising := sReadSDO.SDOData3.LatchCntInput2Rising;
          iDeltaPos := to_int(sLatchValues.uiLatchInputDigIn2Rising - sLatchValues.uiISyncDigIn2RiseOldCounter)/usTempCompMode;
          LatchPositionInput2Rising := sLatchValues.sdISyncDigIn2RiseOldPosition + to_dint(iDeltaPos);
        end_if;
        if sLatchValues.bsValidISyncValue.DigIn2Fall & sReadSDO.SDOData3.LatchCntInput2Falling then
          sLatchValues.uiLatchInputDigIn2Falling := sReadSDO.SDOData3.LatchCntInput2Falling;
          iDeltaPos := to_int(sLatchValues.uiLatchInputDigIn2Falling - sLatchValues.uiISyncDigIn2FallOldCounter)/usTempCompMode;
          LatchPositionInput2Falling := sLatchValues.sdISyncDigIn2FallOldPosition + to_dint(iDeltaPos);
        end_if;

      sLatchValues.bsValidISyncValue := 0;
    end_if;
    bsRespSDOConfigRdWr.ReadConfigSDO3 := FALSE;
  end_if;

END_FUNCTION

FUNCTION VIRTUAL GLOBAL ST151Base::ConnectEvent

  // start the accesses on the SDIAS (initialize the control byte in the DPRAM)
  //Read Access
  if DefaultAccesses.ReadAccess.pControlByte then
    sAccesses.pReadData := DefaultAccesses.ReadAccess.pData$^t_s_ReadData;

    DefaultAccesses.ReadAccess.pControlByte^.EnableDO := TRUE;
  else
    eInitState := _DOHandleInvalid;
    return;
  end_if;

  //Write Access
  if DefaultAccesses.WriteAccess.pControlByte then
    sAccesses.pWriteData := DefaultAccesses.WriteAccess.pData$^t_s_WriteData;

    DefaultAccesses.WriteAccess.pControlByte^.EnableDO := TRUE;
  else
    eInitState := _DOHandleInvalid;
    return;
  end_if;

  if UseOszi then
    if sAccessesOszi.ReadHeaderControl.pControlByte then
      //Start Read-Access to Module (Set ControlWord in DPRam)
      sAccessesOszi.ReadHeaderControl.pControlByte^.EnableDO := true;
    else
      //No ControlWord available
      eInitState := _DOHandleInvalid;
      return;
    end_if;

    //Write Access
    if sAccessesOszi.WriteHeaderControl.pControlByte then
      //Start Write-Access to Module (Set ControlWord in DPRam)
      sAccessesOszi.WriteHeaderControl.pControlByte^.EnableDO := true;
    else
      //No ControlWord available
      eInitState := _DOHandleInvalid;
      return;
    end_if;
  end_if;

  //The writing of the configuration must be deactivated here in order to read the default values of the module first. The desired settings are then written automatically.
  biReqSDOConfigRdWr.WriteConfigSDO1 := FALSE;
  biReqSDOConfigRdWr.WriteConfigSDO2 := FALSE;
  biReqSDOConfigRdWr.WriteConfigSDO3 := FALSE;
  biReqSDOConfigRdWr.WriteConfigSDO4 := FALSE;
  biReqSDOConfigRdWr.WriteConfigSDO5 := FALSE;
  biReqSDOConfigRdWr.WriteConfigSDO6 := FALSE;

  biReqSDOConfigRdWr.ReadConfigSDO1 := TRUE;
  biReqSDOConfigRdWr.ReadConfigSDO2 := TRUE;
  biReqSDOConfigRdWr.ReadConfigSDO3 := TRUE;
  biReqSDOConfigRdWr.ReadConfigSDO4 := TRUE;
  biReqSDOConfigRdWr.ReadConfigSDO5 := TRUE;
  biReqSDOConfigRdWr.ReadConfigSDO6 := TRUE;

  usSDORetrys    := 0;
  eInitSSW       := _ReadInitValuesFromModule;
  eInitState     := _NotInitialized;
  eResponseState := _idle;

END_FUNCTION

FUNCTION VIRTUAL GLOBAL ST151Base::CheckDeviceID
	VAR_INPUT
		udID2Check 	: UDINT;
	END_VAR
	VAR_OUTPUT
		bIsOK 	: BOOL;
	END_VAR

  if (udID2Check <> DEVICE_ID_ST151) then
    bIsOK := FALSE;
  else
    bIsOK := TRUE;
  end_if;

END_FUNCTION

FUNCTION VIRTUAL GLOBAL ST151Base::InitModule
	VAR_OUTPUT
		eModuleInitState 	: iprStates;
	END_VAR
  VAR
  	TmpRetcode      : iprStates;
    hTabAddress : ^UDINT;
  END_VAR

  eModuleInitState := BUSY;

  case eInitSSW of

//**********************************************************************************************************************************************************
    _ReadInitValuesFromModule:
      TmpRetcode := SDORdWrData();
      if TmpRetcode = READY then
        sWriteSDO := sReadSDO;
        eInitSSW  := _InitVariables;
      elsif TmpRetcode = ERROR then
        LogError("@ZZZZ (ST151Base::InitModule) Failed to add read SDO for configuration");
        eInitSSWErrorStep := eInitSSW;
        eInitSSW          := _InitError;
        eInitState        := _NoMem;
      end_if;

//**********************************************************************************************************************************************************
    _InitVariables:
      //Invert Enable Settings
      Enable.Write(Enable); //--- to ensure function of InvertEnable

      // remember flags for further use
      InvertZeroPosition  := InvertZeroPosition.Read() <> 0;
      InvertEncoder       := InvertEncoder.Read() <> 0;
      EncoderSampling     := EncoderSampling.Read();
      EncMode             := EncMode.Read() <> 0;
      ABCountMode         := ABCountMode.Read() <> 0;
      LatchType           := LatchType.Read() <> 0;
      EncoderSampling     := EncoderSampling.Read();

      StallCurrentReduction := StallCurrentReduction.Read();
      StallCurrentWindow    := StallCurrentWindow.Read();
      EnableRegenResistor   := EnableRegenResistor.Read() <> 0;
      RegenResistance       := RegenResistance.Read();
      RatedMaxPower         := RatedMaxPower.Read();
      LoadThresholdWarning  := LoadThresholdWarning.Read();
      LoadThresholdResistor := LoadThresholdResistor.Read();
      LoadThresholdBridge   := LoadThresholdBridge.Read();
      SteppingHysteresis    := SteppingHysteresis.Read();
      CompModeVST           := CompModeVST.Read() <> 0;

      //set value for stepping hysterese
      udLimitsHysteresis := SteppingHysteresis$UDINT;

      //Limit Encoder Sampling
      if ( EncoderSampling < 0 ) then
        EncoderSampling := 0;
      elsif ( EncoderSampling > 3 ) then
        EncoderSampling := 3;
      end_if;

      //Check for Limits
      if StallCurrentReduction < 0 then
        StallCurrentReduction := 0;
      elsif StallCurrentReduction > ST151_STALL_CURRENT_LIMIT then
        StallCurrentReduction := ST151_STALL_CURRENT_LIMIT;
      end_if;

      if StallCurrentWindow > 0 then
        udStallCurrentWindow := StallCurrentWindow$UDINT;
      else
        udStallCurrentWindow := 0;
      end_if;

      MaxCurrent.Write(input:=MaxCurrent);

      //reset incremental encoder register
      sWriteSDO.SDOData2.IncrementalEncoderSettings := 0;
      //Set Mode of Encoder
      sWriteSDO.SDOData2.IncrementalEncoderSettings.TTL_RS422Mode := EncMode <> 0;
      //set virtual or encoder latch type
      sWriteSDO.SDOData2.IncrementalEncoderSettings.LatchType := LatchType <> 0;

      sWriteSDO.SDOData2.IncrementalEncoderSettings.ZeroPosInversion := InvertZeroPosition <> 0;
      sWriteSDO.SDOData2.IncrementalEncoderSettings.PhaseBInversion  := InvertEncoder <> 0;
      //set edge sampling mode
      sWriteSDO.SDOData2.IncrementalEncoderSettings.EdgeSampling1    := EncoderSampling$BOOL;
      sWriteSDO.SDOData2.IncrementalEncoderSettings.EdgeSampling2    := (EncoderSampling shr 1)$BOOL;
      //set A/B count mode
      sWriteSDO.SDOData2.IncrementalEncoderSettings.ABCountMode := ABCountMode <> 0;

      HWRampdownDeltaFrequency.Write(input:=HWRampdownDeltaFrequency);
      HWRampdownDeltaTime.Write(input:=HWRampdownDeltaTime);
      //set compatibilty variable
      usCompModeVST := CompModeVST$USINT + 1;

      ChopperOffTime.Write(input:=ChopperOffTime);
      ChopperOnTimeMin.Write(input:=ChopperOnTimeMin);
      FastDecayTime.Write(input:=FastDecayTime);
      FastDecayTimeFallingStep.Write(input:=FastDecayTimeFallingStep);
      CurrentOffsetAdjBridge1.Write(input:=CurrentOffsetAdjBridge1);
      CurrentOffsetAdjBridge2.Write(input:=CurrentOffsetAdjBridge2);

      //initialize frequency limits increase frequency
      FrequLimitIncrease2to1.Write(input:=FrequLimitIncrease2to1);
      FrequLimitIncrease4to2.Write(input:=FrequLimitIncrease4to2);
      FrequLimitIncrease8to4.Write(input:=FrequLimitIncrease8to4);
      FrequLimitIncrease16to8.Write(input:=FrequLimitIncrease16to8);
      FrequLimitIncrease32to16.Write(input:=FrequLimitIncrease32to16);
      FrequLimitIncrease64to32.Write(input:=FrequLimitIncrease64to32);
      //initialize frequency limits decrease frequency
      FrequLimitDecrease1to2.Write(input:=FrequLimitDecrease1to2);
      FrequLimitDecrease2to4.Write(input:=FrequLimitDecrease2to4);
      FrequLimitDecrease4to8.Write(input:=FrequLimitDecrease4to8);
      FrequLimitDecrease8to16.Write(input:=FrequLimitDecrease8to16);
      FrequLimitDecrease16to32.Write(input:=FrequLimitDecrease16to32);
      FrequLimitDecrease32to64.Write(input:=FrequLimitDecrease32to64);

      if IsClientConnected(#toFreqLimitTable) then
        hTabAddress$DINT := toFreqLimitTable.Read();
        if hTabAddress^ = ST151_FREQLIMITS_TABLESIZE then
          hTabAddress += sizeof(UDINT);
          FrequLimitIncrease64to32.Write(input:=hTabAddress^);
          hTabAddress += sizeof(UDINT);
          FrequLimitDecrease32to64.Write(input:=hTabAddress^);
          hTabAddress += sizeof(UDINT);
          FrequLimitIncrease32to16.Write(input:=hTabAddress^);
          hTabAddress += sizeof(UDINT);
          FrequLimitDecrease16to32.Write(input:=hTabAddress^);
          hTabAddress += sizeof(UDINT);
          FrequLimitIncrease16to8.Write(input:=hTabAddress^);
          hTabAddress += sizeof(UDINT);
          FrequLimitDecrease8to16.Write(input:=hTabAddress^);
          hTabAddress += sizeof(UDINT);
          FrequLimitIncrease8to4.Write(input:=hTabAddress^);
          hTabAddress += sizeof(UDINT);
          FrequLimitDecrease4to8.Write(input:=hTabAddress^);
          hTabAddress += sizeof(UDINT);
          FrequLimitIncrease4to2.Write(input:=hTabAddress^);
          hTabAddress += sizeof(UDINT);
          FrequLimitDecrease2to4.Write(input:=hTabAddress^);
          hTabAddress += sizeof(UDINT);
          FrequLimitIncrease2to1.Write(input:=hTabAddress^);
          hTabAddress += sizeof(UDINT);
          FrequLimitDecrease1to2.Write(input:=hTabAddress^);
        end_if;
      end_if;

      //initialize variable enable
      EnableSteps.Write(input:=EnableSteps+0x800);

      CurrentIncrease.Write(input:=CurrentIncrease);

      if RatedMaxPower > 0xFFFF then
        RatedMaxPower := 0xFFFF;
      elsif RatedMaxPower < 1 then
        RatedMaxPower := 1;
      end_if;
      sWriteSDO.SDOData2.RatedMaximumPowerWatt := RatedMaxPower$UINT;

      if RegenResistance > 0xFFFF then
        RegenResistance := 0xFFFF;
      elsif RegenResistance < 1 then
        RegenResistance := 1;
      end_if;
      sWriteSDO.SDOData2.RegenResistance := RegenResistance$UINT;

      if LoadThresholdWarning > ST151_MAX_ALLOWED_PERCENT then
        LoadThresholdWarning := ST151_MAX_ALLOWED_PERCENT;
      elsif LoadThresholdWarning < 0 then
        LoadThresholdWarning := 0;
      end_if;
      sWriteSDO.SDOData2.LoadThresholdWarning := LoadThresholdWarning$USINT;

      if LoadThresholdResistor > ST151_MAX_ALLOWED_PERCENT then
        LoadThresholdResistor := ST151_MAX_ALLOWED_PERCENT;
      elsif LoadThresholdResistor < 0 then
        LoadThresholdResistor := 0;
      end_if;
      sWriteSDO.SDOData2.LoadThresholdDisableResistor := LoadThresholdResistor$USINT;
      sWriteSDO.SDOData2.BlankingTimeRegister := ST151_BLANKING_TIME;

      if LoadThresholdBridge > ST151_MAX_ALLOWED_PERCENT then
        LoadThresholdBridge := ST151_MAX_ALLOWED_PERCENT;
      elsif LoadThresholdBridge < 0 then
        LoadThresholdBridge := 0;
      end_if;
      sWriteSDO.SDOData2.LoadThresholdDisableBridge := LoadThresholdBridge$USINT;

      //frequency is zero at beginning
      eActStepping := Microstepping_64;

      //reset read write request config sdo
      biReqSDOConfigRdWr := 0;

      sAccesses.sWriteData.ControlWord.RegenResistorEnable := EnableRegenResistor$BOOL;
      //begin move with reduced current.
      sAccesses.sWriteData.ControlWord.SwitchMaxCurrent    := True;

      //Set write of config sdo 1-4, 3 is only read sdo
      biReqSDOConfigRdWr.WriteConfigSDO1 := TRUE;
      biReqSDOConfigRdWr.WriteConfigSDO2 := TRUE;
      biReqSDOConfigRdWr.WriteConfigSDO4 := TRUE;
      biReqSDOConfigRdWr.WriteConfigSDO5 := TRUE;
      biReqSDOConfigRdWr.WriteConfigSDO6 := TRUE;

      //load config new
      sWriteSDO.SDOData5.bsControllerControlReg.LoadConfigNew   := FALSE;
      sWriteSDO.sdodata5.bsControllerControlReg.ControllerReset := FALSE;
      eInitSSW   := _WriteConfigSDO;

//**********************************************************************************************************************************************************
    _WriteConfigSDO:
      TmpRetcode := SDORdWrData();
      if TmpRetcode = READY then
        //Set read of config sdo 1-4
        biReqSDOConfigRdWr.ReadConfigSDO1 := TRUE;
        biReqSDOConfigRdWr.ReadConfigSDO2 := TRUE;
        biReqSDOConfigRdWr.ReadConfigSDO3 := TRUE;
        biReqSDOConfigRdWr.ReadConfigSDO4 := TRUE;
        biReqSDOConfigRdWr.ReadConfigSDO5 := TRUE;
        biReqSDOConfigRdWr.ReadConfigSDO6 := TRUE;
        eInitSSW := _ReadConfigSDO;
      elsif TmpRetcode = ERROR then
        LogError("@ZZZZ (ST151Base::InitModule) Failed to add write SDO for configuration");
        eInitSSWErrorStep := eInitSSW;
        eInitSSW          := _InitError;
        eInitState        := _NoMem;
      end_if;

//**********************************************************************************************************************************************************
    _ReadConfigSDO:
      TmpRetcode := SDORdWrData();
      if TmpRetcode = READY then
        eInitSSW          := _DisablePll;
      elsif TmpRetcode = ERROR then
        LogError("@ZZZZ (ST151Base::InitModule) Failed to add SDO for read configuration");
        eInitSSWErrorStep := eInitSSW;
        eInitSSW          := _InitError;
        eInitState        := _NoMem;
      end_if;

//**********************************************************************************************************************************************************
    _DisablePll:
      case eResponseState of
        //*******************************************************
        _idle:
          sPllRegister.bsStateControlReg := 0;
          TmpRetcode  := StartWriteSDO(hOffset  := ST151_PLL_CONTROL
                                      , usLength:= sizeof(sPllRegister.bsStateControlReg)
                                      , pWriteBuffer:=#sPllRegister.bsStateControlReg$USINT
                                      , eCommand:= SDIAS_SDO_CMD_CTRL_WRITE);
          if TmpRetcode = READY then
            udSDOTimeout  := ops.tAbsolute;
            eResponseState:= _wait;
          elsif TmpRetcode = ERROR then
            LogError("@ZZZZ (ST151Base::InitModule) Failed to add write SDO for channel configuration, step DisablePll");
            eInitSSWErrorStep := eInitSSW;
            eInitSSW          := _InitError;
          end_if;

        //*******************************************************
        _wait:
          // wait for response
          if ((ops.tAbsolute - udSDOTimeout) > ST151_SDO_RESPONSE_TIMEOUT) then
            LogError("@ZZZZ (ST151Base::InitModule) SDO Response timeout, step DisablePll");
            eInitSSWErrorStep := eInitSSW;
            eInitSSW          := _InitError;
          end_if;

        //*******************************************************
        _valid:
          eInitSSW        := _ReadPll;
          eResponseState  := _idle;
      end_case;

//**********************************************************************************************************************************************************
    _ReadPll:
      case eResponseState of
        //*******************************************************
        _idle:
          if sSPIReadData.udReadOffset < sizeof(sPllRegister) then
            sSPIReadData.udReadLength := sizeof(sPllRegister) - sSPIReadData.udReadOffset;
            if sSPIReadData.udReadLength > SDIAS_MAX_SDO_READ_LENGTH then
              sSPIReadData.udReadLength := SDIAS_MAX_SDO_READ_LENGTH;
            end_if;
            TmpRetcode  := StartReadSDO(hOffset   :=ST151_PLL_OFFSET + sSPIReadData.udReadOffset$HINT
                                        , usLength:=sSPIReadData.udReadLength$USINT
                                        , eCommand:=SDIAS_SDO_CMD_CTRL_READ);
            if TmpRetcode = READY then
              udSDOTimeout      := ops.tAbsolute;
              eResponseState    := _wait;
            elsif TmpRetcode = ERROR then
              LogError("@ZZZZ (ST151Base::InitModule) Failed to add read SDO to read pll");
              eInitSSWErrorStep := eInitSSW;
              eInitSSW          := _InitError;
            end_if;
          else
            sSPIReadData.udReadOffset := 0;
            eInitSSW := _Finish;
          end_if;

        //*******************************************************
        _wait:
          // wait for response
          if ((ops.tAbsolute - udSDOTimeout) > SDIAS_SDO_TIMEOUT*2) then
            LogError("@ZZZZ (ST151Base::InitModule) SDO Response timeout read pll");
            eInitSSWErrorStep := eInitSSW;
            eInitSSW          := _InitError;
          end_if;

        //*******************************************************
        _valid:
          sSPIReadData.udReadOffset += sSPIReadData.udReadLength$USINT;
          eResponseState    := _idle;
          eInitSSW          := _SetPll;
      end_case;

//**********************************************************************************************************************************************************
    _SetPll:
      case eResponseState of
        //*******************************************************
        _idle:
          sSPIWriteData.usWriteOffset         := 0;
          sPllRegister.udSystemPerTime        := udBusTime / 10;            // convert to 10*ns
          sPllRegister.bsStateControlReg      := 0;
          sPllRegister.bsStateControlReg.Soft_enable  := 1;
          sPllRegister.usSystemPeriodeDividier        := 1;
          //sPllRegister.CompensationDelay // Keep value
          sPLLRegister.SyncOut0.uiOffset         := 0;
          sPllRegister.SyncOut0.usPeriodMulti    := 1; (*SetPllMultiplier();*)
          sPllRegister.SyncOut0.bsSyncStartDelay := 0;
          sPllRegister.SyncOut0.bsControlState.SyncEnable       := 1;
          sPllRegister.SyncOut0.bsControlState.StartDelayEnable := 0;
          sPllRegister.SyncOut0.bsControlState.SyncSelector     := 1;

          TmpRetcode  := StartWriteSDO(hOffset      :=ST151_PLL_OFFSET + sSPIWriteData.usWriteOffset
                                      , usLength    :=sizeof(sPLLRegister)
                                      , pWriteBuffer:=(#sPLLRegister+sSPIWriteData.usWriteOffset)$^USINT
                                      , eCommand    :=SDIAS_SDO_CMD_CTRL_WRITE);

          if TmpRetcode = READY then
            udSDOTimeout  := ops.tAbsolute;
            eResponseState:= _wait;
          elsif TmpRetcode = ERROR then
            LogError("@ZZZZ (ST151Base::InitModul) Failed to add write SDO in step SetPll");
            eInitState        := _PllError;
            eInitSSWErrorStep := eInitSSW;
            eInitSSW          := _InitError;
          end_if;

        //*******************************************************
        _wait:
          // wait for response
          if ((ops.tAbsolute - udSDOTimeout) > ST151_SDO_RESPONSE_TIMEOUT) then
            LogError("@ZZZZ (ST151Base::InitModul) SDO Response timeout SetPll");
            eInitSSWErrorStep := eInitSSW;
            eInitSSW          := _InitError;
          end_if;

        //*******************************************************
        _valid:
          sSPIReadData.udReadOffset := 0;
          eInitSSW        := _Wait4FPGAReset;
          eResponseState  := _idle;
      end_case;

//**********************************************************************************************************************************************************
    _Wait4FPGAReset:
      eInitSSW      := _ActivateFPGA;

//**********************************************************************************************************************************************************
    _ActivateFPGA:
        eInitSSW     := _Finish;

//**********************************************************************************************************************************************************
    _Finish:
    //set cyclic server to invalid value
//      DC24VOk              := ST151_INVALID_VALUE$DINT;
      bsRespSDOConfigRdWr.ReadConfigSDO3 := FALSE;
      VoltageOKEncoder     := ST151_INVALID_VALUE$DINT;
      HBridgeVoltage       := ST151_INVALID_VALUE$DINT;
      HBridgeTemperature   := ST151_INVALID_VALUE$DINT;
      ExternalEnable1      := ST151_INVALID_VALUE$DINT;
      ExternalEnable2      := ST151_INVALID_VALUE$DINT;
      ActRegenResistorLoad  := ST151_INVALID_VALUE$DINT;
      eInitSSW             := _InitVariables;
      eModuleInitState     := READY;
      eInitState           := _ClassOk;
